LIN {X 0,Y 573.286,Z 217.077,A -85,B 0,C 180,E1 -2331.54,E2 -2331.54} C_VEL
LIN {X 0,Y 573.293,Z 217.075,A -85,B 0,C 180,E1 -2334.371,E2 -2334.371} C_VEL
LIN {X 0,Y 573.307,Z 217.075,A -85,B 0,C 180,E1 -2337.188,E2 -2337.188} C_VEL
LIN {X 0,Y 573.317,Z 217.072,A -85,B 0,C 180,E1 -2339.999,E2 -2339.999} C_VEL
LIN {X 0,Y 573.307,Z 217.074,A -85,B 0,C 180,E1 -2342.809,E2 -2342.809} C_VEL
LIN {X 0,Y 573.288,Z 217.076,A -85,B 0,C 180,E1 -2345.627,E2 -2345.627} C_VEL
LIN {X 0,Y 573.302,Z 217.075,A -85,B 0,C 180,E1 -2348.458,E2 -2348.458} C_VEL
LIN {X 0,Y 573.292,Z 217.075,A -85,B 0,C 180,E1 -2351.31,E2 -2351.31} C_VEL
LIN {X 0,Y 573.273,Z 217.08,A -85,B 0,C 180,E1 -2354.424,E2 -2354.424} C_VEL
LIN {X 0,Y 573.246,Z 217.081,A -85,B 0,C 180,E1 -2357.111,E2 -2357.111} C_VEL
LIN {X 0,Y 573.119,Z 217.099,A -85,B 0,C 180,E1 -2358.591,E2 -2358.591} C_VEL
LIN {X 0,Y 573.089,Z 220.567,A -85,B 0,C 180,E1 -2361.585,E2 -2361.585} C_VEL
LIN {X 0,Y 573.066,Z 223.811,A -85,B 0,C 180,E1 -2364.338,E2 -2364.338} C_VEL
LIN {X 0,Y 572.416,Z 224.562,A -85,B 0,C 180,E1 -2364.919,E2 -2364.919} C_VEL
LIN {X 0,Y 569.55,Z 225.938,A -85,B 0,C 180,E1 -2365.861,E2 -2365.861} C_VEL
LIN {X 0,Y 567.109,Z 227.058,A -85,B 0,C 180,E1 -2366.618,E2 -2366.618} C_VEL
LIN {X 0,Y 566.053,Z 227.855,A -85,B 0,C 180,E1 -2367.204,E2 -2367.204} C_VEL
LIN {X 0,Y 565.963,Z 228.105,A -85,B 0,C 180,E1 -2367.402,E2 -2367.402} C_VEL
LIN {X 0,Y 565.967,Z 230.788,A -85,B 0,C 180,E1 -2369.781,E2 -2369.781} C_VEL
LIN {X 0,Y 565.878,Z 233.608,A -85,B 0,C 180,E1 -2372.379,E2 -2372.379} C_VEL
LIN {X 0,Y 565.833,Z 236.534,A -85,B 0,C 180,E1 -2374.941,E2 -2374.941} C_VEL
LIN {X 0,Y 565.809,Z 239.829,A -85,B 0,C 180,E1 -2377.489,E2 -2377.489} C_VEL
LIN {X 0,Y 565.833,Z 243.678,A -85,B 0,C 180,E1 -2380.428,E2 -2380.428} C_VEL
LIN {X 0,Y 566.887,Z 251.297,A -85,B 0,C 180,E1 -2380.629,E2 -2380.629} C_VEL
LIN {X 0,Y 566.793,Z 264.173,A -85,B 0,C 180,E1 -2381.027,E2 -2381.027} C_VEL
LIN {X 0,Y 566.586,Z 276.718,A -85,B 0,C 180,E1 -2381.574,E2 -2381.574} C_VEL
LIN {X 0,Y 566.487,Z 287.395,A -85,B 0,C 180,E1 -2382.18,E2 -2382.18} C_VEL
LIN {X 0,Y 566.375,Z 298.091,A -85,B 0,C 180,E1 -2382.937,E2 -2382.937} C_VEL
LIN {X 0,Y 566.243,Z 307.919,A -85,B 0,C 180,E1 -2383.797,E2 -2383.797} C_VEL
LIN {X 0,Y 566.107,Z 317.442,A -85,B 0,C 180,E1 -2384.833,E2 -2384.833} C_VEL
LIN {X 0,Y 566.031,Z 325.716,A -85,B 0,C 180,E1 -2385.949,E2 -2385.949} C_VEL
LIN {X 0,Y 565.958,Z 332.481,A -85,B 0,C 180,E1 -2387.107,E2 -2387.107} C_VEL
LIN {X 0,Y 565.935,Z 337.377,A -85,B 0,C 180,E1 -2388.165,E2 -2388.165} C_VEL
LIN {X 0,Y 565.917,Z 341.246,A -85,B 0,C 180,E1 -2389.246,E2 -2389.246} C_VEL
LIN {X 0,Y 565.871,Z 344.136,A -85,B 0,C 180,E1 -2390.354,E2 -2390.354} C_VEL
LIN {X 0,Y 565.847,Z 346.173,A -85,B 0,C 180,E1 -2391.611,E2 -2391.611} C_VEL
LIN {X 0,Y 565.833,Z 346.918,A -85,B 0,C 180,E1 -2392.645,E2 -2392.645} C_VEL
LIN {X 0,Y 565.815,Z 346.733,A -85,B 0,C 180,E1 -2393.836,E2 -2393.836} C_VEL
LIN {X 0,Y 565.847,Z 345.233,A -85,B 0,C 180,E1 -2395.158,E2 -2395.158} C_VEL
LIN {X 0,Y 565.899,Z 342.77,A -85,B 0,C 180,E1 -2396.31,E2 -2396.31} C_VEL
LIN {X 0,Y 565.878,Z 338.598,A -85,B 0,C 180,E1 -2397.619,E2 -2397.619} C_VEL
LIN {X 0,Y 565.944,Z 334.577,A -85,B 0,C 180,E1 -2398.564,E2 -2398.564} C_VEL
LIN {X 0,Y 566.021,Z 329.055,A -85,B 0,C 180,E1 -2399.605,E2 -2399.605} C_VEL
LIN {X 0,Y 566.069,Z 322.304,A -85,B 0,C 180,E1 -2400.633,E2 -2400.633} C_VEL
LIN {X 0,Y 566.159,Z 313.851,A -85,B 0,C 180,E1 -2401.674,E2 -2401.674} C_VEL
LIN {X 0,Y 566.27,Z 303.926,A -85,B 0,C 180,E1 -2402.665,E2 -2402.665} C_VEL
LIN {X 0,Y 566.435,Z 293.893,A -85,B 0,C 180,E1 -2403.471,E2 -2403.471} C_VEL
LIN {X 0,Y 566.508,Z 283.157,A -85,B 0,C 180,E1 -2404.168,E2 -2404.168} C_VEL
LIN {X 0,Y 566.677,Z 271.149,A -85,B 0,C 180,E1 -2404.779,E2 -2404.779} C_VEL
LIN {X 0,Y 566.823,Z 259.841,A -85,B 0,C 180,E1 -2405.214,E2 -2405.214} C_VEL
LIN {X 0,Y 566.718,Z 248.791,A -85,B 0,C 180,E1 -2405.527,E2 -2405.527} C_VEL
LIN {X 0,Y 565.875,Z 243.68,A -85,B 0,C 180,E1 -2405.659,E2 -2405.659} C_VEL
LIN {X 0,Y 565.885,Z 239.45,A -85,B 0,C 180,E1 -2408.89,E2 -2408.89} C_VEL
LIN {X 0,Y 565.873,Z 236.517,A -85,B 0,C 180,E1 -2411.162,E2 -2411.162} C_VEL
LIN {X 0,Y 565.896,Z 233.864,A -85,B 0,C 180,E1 -2413.404,E2 -2413.404} C_VEL
LIN {X 0,Y 565.962,Z 230.528,A -85,B 0,C 180,E1 -2416.354,E2 -2416.354} C_VEL
LIN {X 0,Y 565.958,Z 227.036,A -85,B 0,C 180,E1 -2419.266,E2 -2419.266} C_VEL
LIN {X 0,Y 566.008,Z 223.617,A -85,B 0,C 180,E1 -2422.15,E2 -2422.15} C_VEL
LIN {X 0,Y 566.06,Z 220.337,A -85,B 0,C 180,E1 -2425.015,E2 -2425.015} C_VEL
LIN {X 0,Y 566.002,Z 217.986,A -85,B 0,C 180,E1 -2427.154,E2 -2427.154} C_VEL
LIN {X 0,Y 566.299,Z 217.947,A -85,B 0,C 180,E1 -2429.29,E2 -2429.29} C_VEL
LIN {X 0,Y 566.27,Z 217.949,A -85,B 0,C 180,E1 -2432.135,E2 -2432.135} C_VEL
LIN {X 0,Y 566.251,Z 217.952,A -85,B 0,C 180,E1 -2435.699,E2 -2435.699} C_VEL
LIN {X 0,Y 566.238,Z 217.955,A -85,B 0,C 180,E1 -2438.566,E2 -2438.566} C_VEL
LIN {X 0,Y 566.238,Z 217.953,A -85,B 0,C 180,E1 -2441.455,E2 -2441.455} C_VEL
LIN {X 0,Y 566.221,Z 217.957,A -85,B 0,C 180,E1 -2444.508,E2 -2444.508} C_VEL
LIN {X 0,Y 566.193,Z 217.959,A -85,B 0,C 180,E1 -2447.333,E2 -2447.333} C_VEL
LIN {X 0,Y 566.21,Z 217.958,A -85,B 0,C 180,E1 -2450.338,E2 -2450.338} C_VEL
LIN {X 0,Y 566.219,Z 217.958,A -85,B 0,C 180,E1 -2453.403,E2 -2453.403} C_VEL
LIN {X 0,Y 566.217,Z 217.958,A -85,B 0,C 180,E1 -2455.75,E2 -2455.75} C_VEL
LIN {X 0,Y 566.199,Z 217.96,A -85,B 0,C 180,E1 -2458.205,E2 -2458.205} C_VEL
LIN {X 0,Y 566.19,Z 217.96,A -85,B 0,C 180,E1 -2461.08,E2 -2461.08} C_VEL
LIN {X 0,Y 566.221,Z 217.958,A -85,B 0,C 180,E1 -2463.739,E2 -2463.739} C_VEL
LIN {X 0,Y 566.209,Z 217.957,A -85,B 0,C 180,E1 -2466.57,E2 -2466.57} C_VEL
LIN {X 0,Y 566.207,Z 217.959,A -85,B 0,C 180,E1 -2469.687,E2 -2469.687} C_VEL
LIN {X 0,Y 566.211,Z 217.958,A -85,B 0,C 180,E1 -2472.088,E2 -2472.088} C_VEL
LIN {X 0,Y 566.167,Z 217.964,A -85,B 0,C 180,E1 -2475.037,E2 -2475.037} C_VEL
LIN {X 0,Y 566.213,Z 217.956,A -85,B 0,C 180,E1 -2478.137,E2 -2478.137} C_VEL
LIN {X 0,Y 566.22,Z 217.957,A -85,B 0,C 180,E1 -2480.729,E2 -2480.729} C_VEL
LIN {X 0,Y 566.212,Z 217.956,A -85,B 0,C 180,E1 -2483.785,E2 -2483.785} C_VEL
LIN {X 0,Y 566.227,Z 217.955,A -85,B 0,C 180,E1 -2486.9,E2 -2486.9} C_VEL
LIN {X 0,Y 566.18,Z 217.96,A -85,B 0,C 180,E1 -2489.409,E2 -2489.409} C_VEL
LIN {X 0,Y 566.211,Z 217.957,A -85,B 0,C 180,E1 -2491.859,E2 -2491.859} C_VEL
LIN {X 0,Y 566.215,Z 217.956,A -85,B 0,C 180,E1 -2494.253,E2 -2494.253} C_VEL
LIN {X 0,Y 566.17,Z 217.963,A -85,B 0,C 180,E1 -2496.721,E2 -2496.721} C_VEL
LIN {X 0,Y 566.217,Z 217.956,A -85,B 0,C 180,E1 -2499.664,E2 -2499.664} C_VEL
LIN {X 0,Y 566.202,Z 217.96,A -85,B 0,C 180,E1 -2502.67,E2 -2502.67} C_VEL
LIN {X 0,Y 566.238,Z 217.953,A -85,B 0,C 180,E1 -2505.628,E2 -2505.628} C_VEL
LIN {X 0,Y 566.239,Z 217.953,A -85,B 0,C 180,E1 -2508.677,E2 -2508.677} C_VEL
LIN {X 0,Y 566.211,Z 217.957,A -85,B 0,C 180,E1 -2511.435,E2 -2511.435} C_VEL
LIN {X 0,Y 566.216,Z 217.956,A -85,B 0,C 180,E1 -2513.587,E2 -2513.587} C_VEL
LIN {X 0,Y 566.187,Z 217.96,A -85,B 0,C 180,E1 -2515.73,E2 -2515.73} C_VEL
LIN {X 0,Y 566.276,Z 217.949,A -85,B 0,C 180,E1 -2517.867,E2 -2517.867} C_VEL
LIN {X 0,Y 566.302,Z 217.946,A -85,B 0,C 180,E1 -2520.712,E2 -2520.712} C_VEL
LIN {X 0,Y 566.271,Z 217.948,A -85,B 0,C 180,E1 -2522.847,E2 -2522.847} C_VEL
LIN {X 0,Y 566.258,Z 217.953,A -85,B 0,C 180,E1 -2525.699,E2 -2525.699} C_VEL
LIN {X 0,Y 566.212,Z 217.956,A -85,B 0,C 180,E1 -2528.567,E2 -2528.567} C_VEL
LIN {X 0,Y 566.25,Z 217.954,A -85,B 0,C 180,E1 -2531.455,E2 -2531.455} C_VEL
LIN {X 0,Y 566.227,Z 217.955,A -85,B 0,C 180,E1 -2534.501,E2 -2534.501} C_VEL
LIN {X 0,Y 566.198,Z 217.959,A -85,B 0,C 180,E1 -2537.333,E2 -2537.333} C_VEL
LIN {X 0,Y 566.216,Z 217.958,A -85,B 0,C 180,E1 -2540.338,E2 -2540.338} C_VEL
LIN {X 0,Y 566.175,Z 217.961,A -85,B 0,C 180,E1 -2543.281,E2 -2543.281} C_VEL
LIN {X 0,Y 566.211,Z 217.957,A -85,B 0,C 180,E1 -2545.75,E2 -2545.75} C_VEL
LIN {X 0,Y 566.212,Z 217.957,A -85,B 0,C 180,E1 -2548.202,E2 -2548.202} C_VEL
LIN {X 0,Y 566.194,Z 217.96,A -85,B 0,C 180,E1 -2551.076,E2 -2551.076} C_VEL
LIN {X 0,Y 566.205,Z 217.957,A -85,B 0,C 180,E1 -2553.732,E2 -2553.732} C_VEL
LIN {X 0,Y 566.208,Z 217.96,A -85,B 0,C 180,E1 -2556.57,E2 -2556.57} C_VEL
LIN {X 0,Y 566.221,Z 217.957,A -85,B 0,C 180,E1 -2559.686,E2 -2559.686} C_VEL
LIN {X 0,Y 566.21,Z 217.957,A -85,B 0,C 180,E1 -2562.917,E2 -2562.917} C_VEL
LIN {X 0,Y 566.202,Z 217.957,A -85,B 0,C 180,E1 -2566.049,E2 -2566.049} C_VEL
LIN {X 0,Y 566.212,Z 217.958,A -85,B 0,C 180,E1 -2569.214,E2 -2569.214} C_VEL
LIN {X 0,Y 566.189,Z 217.962,A -85,B 0,C 180,E1 -2571.636,E2 -2571.636} C_VEL
LIN {X 0,Y 566.229,Z 218.104,A -85,B 0,C 180,E1 -2573.043,E2 -2573.043} C_VEL
LIN {X 0,Y 566.784,Z 221.774,A -85,B 0,C 180,E1 -2574.352,E2 -2574.352} C_VEL
LIN {X 0,Y 566.714,Z 229.498,A -85,B 0,C 180,E1 -2576.93,E2 -2576.93} C_VEL
LIN {X 0,Y 566.515,Z 237.229,A -85,B 0,C 180,E1 -2579.426,E2 -2579.426} C_VEL
LIN {X 0,Y 566.446,Z 245.3,A -85,B 0,C 180,E1 -2581.869,E2 -2581.869} C_VEL
LIN {X 0,Y 566.345,Z 255.739,A -85,B 0,C 180,E1 -2584.944,E2 -2584.944} C_VEL
LIN {X 0,Y 566.292,Z 265.468,A -85,B 0,C 180,E1 -2587.757,E2 -2587.757} C_VEL
LIN {X 0,Y 566.209,Z 275.582,A -85,B 0,C 180,E1 -2590.622,E2 -2590.622} C_VEL
LIN {X 0,Y 566.129,Z 285.461,A -85,B 0,C 180,E1 -2593.409,E2 -2593.409} C_VEL
LIN {X 0,Y 566.046,Z 296.052,A -85,B 0,C 180,E1 -2596.354,E2 -2596.354} C_VEL
LIN {X 0,Y 566.015,Z 299.528,A -85,B 0,C 180,E1 -2597.313,E2 -2597.313} C_VEL
LIN {X 0,Y 566.935,Z 306.333,A -85,B 0,C 180,E1 -2597.47,E2 -2597.47} C_VEL
LIN {X 0,Y 566.844,Z 318.476,A -85,B 0,C 180,E1 -2597.786,E2 -2597.786} C_VEL
LIN {X 0,Y 566.689,Z 330.299,A -85,B 0,C 180,E1 -2598.228,E2 -2598.228} C_VEL
LIN {X 0,Y 566.534,Z 342.971,A -85,B 0,C 180,E1 -2598.867,E2 -2598.867} C_VEL
LIN {X 0,Y 566.439,Z 354.736,A -85,B 0,C 180,E1 -2599.635,E2 -2599.635} C_VEL
LIN {X 0,Y 566.302,Z 363.639,A -85,B 0,C 180,E1 -2600.355,E2 -2600.355} C_VEL
LIN {X 0,Y 566.162,Z 372.78,A -85,B 0,C 180,E1 -2601.253,E2 -2601.253} C_VEL
LIN {X 0,Y 566.082,Z 381.684,A -85,B 0,C 180,E1 -2602.33,E2 -2602.33} C_VEL
LIN {X 0,Y 565.969,Z 388.952,A -85,B 0,C 180,E1 -2603.422,E2 -2603.422} C_VEL
LIN {X 0,Y 566.004,Z 393.676,A -85,B 0,C 180,E1 -2604.298,E2 -2604.298} C_VEL
LIN {X 0,Y 565.933,Z 398.369,A -85,B 0,C 180,E1 -2605.369,E2 -2605.369} C_VEL
LIN {X 0,Y 565.927,Z 401.956,A -85,B 0,C 180,E1 -2606.439,E2 -2606.439} C_VEL
LIN {X 0,Y 565.878,Z 403.806,A -85,B 0,C 180,E1 -2607.152,E2 -2607.152} C_VEL
LIN {X 0,Y 565.846,Z 406.184,A -85,B 0,C 180,E1 -2608.576,E2 -2608.576} C_VEL
LIN {X 0,Y 565.839,Z 407,A -85,B 0,C 180,E1 -2609.999,E2 -2609.999} C_VEL
LIN {X 0,Y 565.846,Z 406.187,A -85,B 0,C 180,E1 -2611.423,E2 -2611.423} C_VEL
LIN {X 0,Y 565.878,Z 403.812,A -85,B 0,C 180,E1 -2612.847,E2 -2612.847} C_VEL
LIN {X 0,Y 565.926,Z 400.898,A -85,B 0,C 180,E1 -2613.916,E2 -2613.916} C_VEL
LIN {X 0,Y 565.878,Z 396.952,A -85,B 0,C 180,E1 -2614.987,E2 -2614.987} C_VEL
LIN {X 0,Y 566.002,Z 391.871,A -85,B 0,C 180,E1 -2616.058,E2 -2616.058} C_VEL
LIN {X 0,Y 566.04,Z 385.473,A -85,B 0,C 180,E1 -2617.132,E2 -2617.132} C_VEL
LIN {X 0,Y 566.133,Z 377.484,A -85,B 0,C 180,E1 -2618.207,E2 -2618.207} C_VEL
LIN {X 0,Y 566.229,Z 369.342,A -85,B 0,C 180,E1 -2619.105,E2 -2619.105} C_VEL
LIN {X 0,Y 566.348,Z 359.409,A -85,B 0,C 180,E1 -2620.004,E2 -2620.004} C_VEL
LIN {X 0,Y 566.502,Z 348.334,A -85,B 0,C 180,E1 -2620.805,E2 -2620.805} C_VEL
LIN {X 0,Y 566.608,Z 335.96,A -85,B 0,C 180,E1 -2621.509,E2 -2621.509} C_VEL
LIN {X 0,Y 566.749,Z 323.789,A -85,B 0,C 180,E1 -2622.033,E2 -2622.033} C_VEL
LIN {X 0,Y 566.928,Z 310.377,A -85,B 0,C 180,E1 -2622.438,E2 -2622.438} C_VEL
LIN {X 0,Y 566.641,Z 303.554,A -85,B 0,C 180,E1 -2622.592,E2 -2622.592} C_VEL
LIN {X 0,Y 566.014,Z 299.533,A -85,B 0,C 180,E1 -2622.686,E2 -2622.686} C_VEL
LIN {X 0,Y 566.089,Z 289.438,A -85,B 0,C 180,E1 -2625.48,E2 -2625.48} C_VEL
LIN {X 0,Y 566.175,Z 278.847,A -85,B 0,C 180,E1 -2628.453,E2 -2628.453} C_VEL
LIN {X 0,Y 566.237,Z 269.442,A -85,B 0,C 180,E1 -2631.096,E2 -2631.096} C_VEL
LIN {X 0,Y 566.278,Z 259.722,A -85,B 0,C 180,E1 -2633.787,E2 -2633.787} C_VEL
LIN {X 0,Y 566.331,Z 250.15,A -85,B 0,C 180,E1 -2636.534,E2 -2636.534} C_VEL
LIN {X 0,Y 566.468,Z 241.095,A -85,B 0,C 180,E1 -2639.33,E2 -2639.33} C_VEL
LIN {X 0,Y 566.63,Z 231.929,A -85,B 0,C 180,E1 -2642.23,E2 -2642.23} C_VEL
LIN {X 0,Y 566.775,Z 224.253,A -85,B 0,C 180,E1 -2644.777,E2 -2644.777} C_VEL
LIN {X 0,Y 566.551,Z 220.044,A -85,B 0,C 180,E1 -2646.261,E2 -2646.261} C_VEL
LIN {X 0,Y 566.205,Z 217.959,A -85,B 0,C 180,E1 -2647.109,E2 -2647.109} C_VEL
LIN {X 0,Y 566.212,Z 217.959,A -85,B 0,C 180,E1 -2649.685,E2 -2649.685} C_VEL
LIN {X 0,Y 566.214,Z 217.959,A -85,B 0,C 180,E1 -2652.086,E2 -2652.086} C_VEL
LIN {X 0,Y 566.167,Z 217.963,A -85,B 0,C 180,E1 -2655.035,E2 -2655.035} C_VEL
LIN {X 0,Y 566.218,Z 217.956,A -85,B 0,C 180,E1 -2658.135,E2 -2658.135} C_VEL
LIN {X 0,Y 566.215,Z 217.957,A -85,B 0,C 180,E1 -2660.726,E2 -2660.726} C_VEL
LIN {X 0,Y 566.202,Z 217.958,A -85,B 0,C 180,E1 -2663.784,E2 -2663.784} C_VEL
LIN {X 0,Y 566.211,Z 217.957,A -85,B 0,C 180,E1 -2666.265,E2 -2666.265} C_VEL
LIN {X 0,Y 566.187,Z 217.962,A -85,B 0,C 180,E1 -2668.923,E2 -2668.923} C_VEL
LIN {X 0,Y 566.226,Z 217.955,A -85,B 0,C 180,E1 -2671.857,E2 -2671.857} C_VEL
LIN {X 0,Y 566.212,Z 217.957,A -85,B 0,C 180,E1 -2674.25,E2 -2674.25} C_VEL
LIN {X 0,Y 566.166,Z 217.963,A -85,B 0,C 180,E1 -2676.718,E2 -2676.718} C_VEL
LIN {X 0,Y 566.211,Z 217.957,A -85,B 0,C 180,E1 -2679.662,E2 -2679.662} C_VEL
LIN {X 0,Y 566.197,Z 217.961,A -85,B 0,C 180,E1 -2682.667,E2 -2682.667} C_VEL
LIN {X 0,Y 566.231,Z 217.954,A -85,B 0,C 180,E1 -2685.626,E2 -2685.626} C_VEL
LIN {X 0,Y 566.23,Z 217.954,A -85,B 0,C 180,E1 -2688.674,E2 -2688.674} C_VEL
LIN {X 0,Y 566.229,Z 217.955,A -85,B 0,C 180,E1 -2691.433,E2 -2691.433} C_VEL
LIN {X 0,Y 566.26,Z 217.951,A -85,B 0,C 180,E1 -2694.301,E2 -2694.301} C_VEL
LIN {X 0,Y 566.271,Z 217.949,A -85,B 0,C 180,E1 -2697.865,E2 -2697.865} C_VEL
LIN {X 0,Y 566.304,Z 217.948,A -85,B 0,C 180,E1 -2700.71,E2 -2700.71} C_VEL
LIN {X 0,Y 566.272,Z 217.951,A -85,B 0,C 180,E1 -2702.844,E2 -2702.844} C_VEL
LIN {X 0,Y 566.256,Z 217.951,A -85,B 0,C 180,E1 -2705.697,E2 -2705.697} C_VEL
LIN {X 0,Y 566.243,Z 217.955,A -85,B 0,C 180,E1 -2708.564,E2 -2708.564} C_VEL
LIN {X 0,Y 566.244,Z 217.953,A -85,B 0,C 180,E1 -2711.453,E2 -2711.453} C_VEL
LIN {X 0,Y 566.226,Z 217.957,A -85,B 0,C 180,E1 -2714.506,E2 -2714.506} C_VEL
LIN {X 0,Y 566.178,Z 217.962,A -85,B 0,C 180,E1 -2717.331,E2 -2717.331} C_VEL
LIN {X 0,Y 566.055,Z 218.047,A -85,B 0,C 180,E1 -2718.831,E2 -2718.831} C_VEL
LIN {X 0,Y 566.049,Z 220.993,A -85,B 0,C 180,E1 -2721.381,E2 -2721.381} C_VEL
LIN {X 0,Y 565.99,Z 224.427,A -85,B 0,C 180,E1 -2724.331,E2 -2724.331} C_VEL
LIN {X 0,Y 565.985,Z 227.149,A -85,B 0,C 180,E1 -2726.616,E2 -2726.616} C_VEL
LIN {X 0,Y 565.963,Z 228.105,A -85,B 0,C 180,E1 -2727.402,E2 -2727.402} C_VEL
LIN {X 0,Y 565.283,Z 228.882,A -85,B 0,C 180,E1 -2727.991,E2 -2727.991} C_VEL
LIN {X 0,Y 562.408,Z 230.258,A -85,B 0,C 180,E1 -2728.946,E2 -2728.946} C_VEL
LIN {X 0,Y 559.98,Z 231.306,A -85,B 0,C 180,E1 -2729.715,E2 -2729.715} C_VEL
LIN {X 0,Y 558.934,Z 232.024,A -85,B 0,C 180,E1 -2730.31,E2 -2730.31} C_VEL
LIN {X 0,Y 558.847,Z 232.245,A -85,B 0,C 180,E1 -2730.511,E2 -2730.511} C_VEL
LIN {X 0,Y 558.809,Z 235.592,A -85,B 0,C 180,E1 -2733.597,E2 -2733.597} C_VEL
LIN {X 0,Y 558.731,Z 238.749,A -85,B 0,C 180,E1 -2736.389,E2 -2736.389} C_VEL
LIN {X 0,Y 558.713,Z 241.999,A -85,B 0,C 180,E1 -2738.97,E2 -2738.97} C_VEL
LIN {X 0,Y 558.751,Z 243.681,A -85,B 0,C 180,E1 -2740.268,E2 -2740.268} C_VEL
LIN {X 0,Y 559.962,Z 252.449,A -85,B 0,C 180,E1 -2740.502,E2 -2740.502} C_VEL
LIN {X 0,Y 559.843,Z 264.145,A -85,B 0,C 180,E1 -2740.874,E2 -2740.874} C_VEL
LIN {X 0,Y 559.631,Z 276.024,A -85,B 0,C 180,E1 -2741.394,E2 -2741.394} C_VEL
LIN {X 0,Y 559.492,Z 288.404,A -85,B 0,C 180,E1 -2742.107,E2 -2742.107} C_VEL
LIN {X 0,Y 559.361,Z 298.544,A -85,B 0,C 180,E1 -2742.845,E2 -2742.845} C_VEL
LIN {X 0,Y 559.202,Z 308.372,A -85,B 0,C 180,E1 -2743.726,E2 -2743.726} C_VEL
LIN {X 0,Y 559.064,Z 317.573,A -85,B 0,C 180,E1 -2744.745,E2 -2744.745} C_VEL
LIN {X 0,Y 558.978,Z 325.16,A -85,B 0,C 180,E1 -2745.777,E2 -2745.777} C_VEL
LIN {X 0,Y 558.88,Z 332.471,A -85,B 0,C 180,E1 -2747.029,E2 -2747.029} C_VEL
LIN {X 0,Y 558.838,Z 337.762,A -85,B 0,C 180,E1 -2748.201,E2 -2748.201} C_VEL
LIN {X 0,Y 558.825,Z 341.134,A -85,B 0,C 180,E1 -2749.159,E2 -2749.159} C_VEL
LIN {X 0,Y 558.785,Z 343.669,A -85,B 0,C 180,E1 -2750.102,E2 -2750.102} C_VEL
LIN {X 0,Y 558.741,Z 345.757,A -85,B 0,C 180,E1 -2751.244,E2 -2751.244} C_VEL
LIN {X 0,Y 558.74,Z 346.842,A -85,B 0,C 180,E1 -2752.411,E2 -2752.411} C_VEL
LIN {X 0,Y 558.719,Z 346.79,A -85,B 0,C 180,E1 -2753.759,E2 -2753.759} C_VEL
LIN {X 0,Y 558.746,Z 345.764,A -85,B 0,C 180,E1 -2754.84,E2 -2754.84} C_VEL
LIN {X 0,Y 558.793,Z 343.38,A -85,B 0,C 180,E1 -2756.105,E2 -2756.105} C_VEL
LIN {X 0,Y 558.788,Z 339.514,A -85,B 0,C 180,E1 -2757.42,E2 -2757.42} C_VEL
LIN {X 0,Y 558.848,Z 335.296,A -85,B 0,C 180,E1 -2758.473,E2 -2758.473} C_VEL
LIN {X 0,Y 558.935,Z 329.569,A -85,B 0,C 180,E1 -2759.597,E2 -2759.597} C_VEL
LIN {X 0,Y 558.988,Z 322.953,A -85,B 0,C 180,E1 -2760.638,E2 -2760.638} C_VEL
LIN {X 0,Y 559.093,Z 314.66,A -85,B 0,C 180,E1 -2761.693,E2 -2761.693} C_VEL
LIN {X 0,Y 559.238,Z 304.878,A -85,B 0,C 180,E1 -2762.698,E2 -2762.698} C_VEL
LIN {X 0,Y 559.425,Z 295.081,A -85,B 0,C 180,E1 -2763.515,E2 -2763.515} C_VEL
LIN {X 0,Y 559.522,Z 284.646,A -85,B 0,C 180,E1 -2764.221,E2 -2764.221} C_VEL
LIN {X 0,Y 559.711,Z 272.626,A -85,B 0,C 180,E1 -2764.858,E2 -2764.858} C_VEL
LIN {X 0,Y 559.877,Z 260.858,A -85,B 0,C 180,E1 -2765.332,E2 -2765.332} C_VEL
LIN {X 0,Y 559.73,Z 249.375,A -85,B 0,C 180,E1 -2765.671,E2 -2765.671} C_VEL
LIN {X 0,Y 558.776,Z 243.677,A -85,B 0,C 180,E1 -2765.824,E2 -2765.824} C_VEL
LIN {X 0,Y 558.764,Z 240.078,A -85,B 0,C 180,E1 -2768.608,E2 -2768.608} C_VEL
LIN {X 0,Y 558.805,Z 237.294,A -85,B 0,C 180,E1 -2770.914,E2 -2770.914} C_VEL
LIN {X 0,Y 558.831,Z 234.671,A -85,B 0,C 180,E1 -2773.188,E2 -2773.188} C_VEL
LIN {X 0,Y 558.891,Z 231.28,A -85,B 0,C 180,E1 -2776.178,E2 -2776.178} C_VEL
LIN {X 0,Y 558.904,Z 227.787,A -85,B 0,C 180,E1 -2779.129,E2 -2779.129} C_VEL
LIN {X 0,Y 558.936,Z 224.358,A -85,B 0,C 180,E1 -2782.051,E2 -2782.051} C_VEL
LIN {X 0,Y 559.004,Z 221.058,A -85,B 0,C 180,E1 -2784.952,E2 -2784.952} C_VEL
LIN {X 0,Y 558.933,Z 219.387,A -85,B 0,C 180,E1 -2786.396,E2 -2786.396} C_VEL
LIN {X 0,Y 558.949,Z 218.865,A -85,B 0,C 180,E1 -2787.118,E2 -2787.118} C_VEL
LIN {X 0,Y 559.158,Z 218.836,A -85,B 0,C 180,E1 -2788.56,E2 -2788.56} C_VEL
LIN {X 0,Y 559.268,Z 218.824,A -85,B 0,C 180,E1 -2790.721,E2 -2790.721} C_VEL
LIN {X 0,Y 559.229,Z 218.829,A -85,B 0,C 180,E1 -2792.882,E2 -2792.882} C_VEL
LIN {X 0,Y 559.22,Z 218.827,A -85,B 0,C 180,E1 -2795.771,E2 -2795.771} C_VEL
LIN {X 0,Y 559.193,Z 218.834,A -85,B 0,C 180,E1 -2798.675,E2 -2798.675} C_VEL
LIN {X 0,Y 559.196,Z 218.831,A -85,B 0,C 180,E1 -2801.601,E2 -2801.601} C_VEL
LIN {X 0,Y 559.186,Z 218.833,A -85,B 0,C 180,E1 -2804.597,E2 -2804.597} C_VEL
LIN {X 0,Y 559.152,Z 218.837,A -85,B 0,C 180,E1 -2807.558,E2 -2807.558} C_VEL
LIN {X 0,Y 559.164,Z 218.836,A -85,B 0,C 180,E1 -2809.838,E2 -2809.838} C_VEL
LIN {X 0,Y 559.145,Z 218.838,A -85,B 0,C 180,E1 -2812.153,E2 -2812.153} C_VEL
LIN {X 0,Y 559.149,Z 218.838,A -85,B 0,C 180,E1 -2814.506,E2 -2814.506} C_VEL
LIN {X 0,Y 559.171,Z 218.837,A -85,B 0,C 180,E1 -2816.903,E2 -2816.903} C_VEL
LIN {X 0,Y 559.14,Z 218.837,A -85,B 0,C 180,E1 -2819.859,E2 -2819.859} C_VEL
LIN {X 0,Y 559.167,Z 218.837,A -85,B 0,C 180,E1 -2822.715,E2 -2822.715} C_VEL
LIN {X 0,Y 559.151,Z 218.836,A -85,B 0,C 180,E1 -2825.323,E2 -2825.323} C_VEL
LIN {X 0,Y 559.127,Z 218.839,A -85,B 0,C 180,E1 -2828.019,E2 -2828.019} C_VEL
LIN {X 0,Y 559.17,Z 218.835,A -85,B 0,C 180,E1 -2830.812,E2 -2830.812} C_VEL
LIN {X 0,Y 559.158,Z 218.835,A -85,B 0,C 180,E1 -2833.733,E2 -2833.733} C_VEL
LIN {X 0,Y 559.141,Z 218.838,A -85,B 0,C 180,E1 -2836.805,E2 -2836.805} C_VEL
LIN {X 0,Y 559.172,Z 218.833,A -85,B 0,C 180,E1 -2839.191,E2 -2839.191} C_VEL
LIN {X 0,Y 559.132,Z 218.84,A -85,B 0,C 180,E1 -2841.984,E2 -2841.984} C_VEL
LIN {X 0,Y 559.147,Z 218.837,A -85,B 0,C 180,E1 -2844.786,E2 -2844.786} C_VEL
LIN {X 0,Y 559.171,Z 218.833,A -85,B 0,C 180,E1 -2847.363,E2 -2847.363} C_VEL
LIN {X 0,Y 559.148,Z 218.839,A -85,B 0,C 180,E1 -2850.144,E2 -2850.144} C_VEL
LIN {X 0,Y 559.169,Z 218.833,A -85,B 0,C 180,E1 -2853.099,E2 -2853.099} C_VEL
LIN {X 0,Y 559.156,Z 218.835,A -85,B 0,C 180,E1 -2855.496,E2 -2855.496} C_VEL
LIN {X 0,Y 559.174,Z 218.833,A -85,B 0,C 180,E1 -2858.625,E2 -2858.625} C_VEL
LIN {X 0,Y 559.169,Z 218.833,A -85,B 0,C 180,E1 -2860.928,E2 -2860.928} C_VEL
LIN {X 0,Y 559.165,Z 218.837,A -85,B 0,C 180,E1 -2863.949,E2 -2863.949} C_VEL
LIN {X 0,Y 559.175,Z 218.836,A -85,B 0,C 180,E1 -2866.186,E2 -2866.186} C_VEL
LIN {X 0,Y 559.197,Z 218.83,A -85,B 0,C 180,E1 -2869.135,E2 -2869.135} C_VEL
LIN {X 0,Y 559.196,Z 218.832,A -85,B 0,C 180,E1 -2872.055,E2 -2872.055} C_VEL
LIN {X 0,Y 559.256,Z 218.823,A -85,B 0,C 180,E1 -2874.955,E2 -2874.955} C_VEL
LIN {X 0,Y 559.249,Z 218.825,A -85,B 0,C 180,E1 -2877.841,E2 -2877.841} C_VEL
LIN {X 0,Y 559.273,Z 218.821,A -85,B 0,C 180,E1 -2880.721,E2 -2880.721} C_VEL
LIN {X 0,Y 559.239,Z 218.824,A -85,B 0,C 180,E1 -2882.882,E2 -2882.882} C_VEL
LIN {X 0,Y 559.228,Z 218.828,A -85,B 0,C 180,E1 -2885.771,E2 -2885.771} C_VEL
LIN {X 0,Y 559.176,Z 218.833,A -85,B 0,C 180,E1 -2888.676,E2 -2888.676} C_VEL
LIN {X 0,Y 559.213,Z 218.829,A -85,B 0,C 180,E1 -2891.601,E2 -2891.601} C_VEL
LIN {X 0,Y 559.19,Z 218.833,A -85,B 0,C 180,E1 -2894.588,E2 -2894.588} C_VEL
LIN {X 0,Y 559.143,Z 218.837,A -85,B 0,C 180,E1 -2897.558,E2 -2897.558} C_VEL
LIN {X 0,Y 559.175,Z 218.833,A -85,B 0,C 180,E1 -2899.838,E2 -2899.838} C_VEL
LIN {X 0,Y 559.148,Z 218.836,A -85,B 0,C 180,E1 -2902.153,E2 -2902.153} C_VEL
LIN {X 0,Y 559.148,Z 218.838,A -85,B 0,C 180,E1 -2905.178,E2 -2905.178} C_VEL
LIN {X 0,Y 559.15,Z 218.836,A -85,B 0,C 180,E1 -2907.715,E2 -2907.715} C_VEL
LIN {X 0,Y 559.157,Z 218.834,A -85,B 0,C 180,E1 -2910.183,E2 -2910.183} C_VEL
LIN {X 0,Y 559.159,Z 218.835,A -85,B 0,C 180,E1 -2912.716,E2 -2912.716} C_VEL
LIN {X 0,Y 559.136,Z 218.841,A -85,B 0,C 180,E1 -2915.324,E2 -2915.324} C_VEL
LIN {X 0,Y 559.138,Z 218.837,A -85,B 0,C 180,E1 -2918.018,E2 -2918.018} C_VEL
LIN {X 0,Y 559.164,Z 218.835,A -85,B 0,C 180,E1 -2920.813,E2 -2920.813} C_VEL
LIN {X 0,Y 559.146,Z 218.837,A -85,B 0,C 180,E1 -2923.734,E2 -2923.734} C_VEL
LIN {X 0,Y 559.153,Z 218.838,A -85,B 0,C 180,E1 -2926.804,E2 -2926.804} C_VEL
LIN {X 0,Y 559.164,Z 218.836,A -85,B 0,C 180,E1 -2929.187,E2 -2929.187} C_VEL
LIN {X 0,Y 559.137,Z 218.839,A -85,B 0,C 180,E1 -2931.982,E2 -2931.982} C_VEL
LIN {X 0,Y 559.162,Z 218.929,A -85,B 0,C 180,E1 -2932.795,E2 -2932.795} C_VEL
LIN {X 0,Y 559.821,Z 223.042,A -85,B 0,C 180,E1 -2934.284,E2 -2934.284} C_VEL
LIN {X 0,Y 559.741,Z 230.761,A -85,B 0,C 180,E1 -2936.894,E2 -2936.894} C_VEL
LIN {X 0,Y 559.537,Z 238.487,A -85,B 0,C 180,E1 -2939.422,E2 -2939.422} C_VEL
LIN {X 0,Y 559.43,Z 246.661,A -85,B 0,C 180,E1 -2941.933,E2 -2941.933} C_VEL
LIN {X 0,Y 559.345,Z 256.197,A -85,B 0,C 180,E1 -2944.778,E2 -2944.778} C_VEL
LIN {X 0,Y 559.217,Z 265.249,A -85,B 0,C 180,E1 -2947.46,E2 -2947.46} C_VEL
LIN {X 0,Y 559.147,Z 274.67,A -85,B 0,C 180,E1 -2950.161,E2 -2950.161} C_VEL
LIN {X 0,Y 559.083,Z 284.139,A -85,B 0,C 180,E1 -2952.818,E2 -2952.818} C_VEL
LIN {X 0,Y 558.986,Z 293.602,A -85,B 0,C 180,E1 -2955.491,E2 -2955.491} C_VEL
LIN {X 0,Y 558.94,Z 299.528,A -85,B 0,C 180,E1 -2957.149,E2 -2957.149} C_VEL
LIN {X 0,Y 560.017,Z 307.473,A -85,B 0,C 180,E1 -2957.336,E2 -2957.336} C_VEL
LIN {X 0,Y 559.878,Z 319.854,A -85,B 0,C 180,E1 -2957.678,E2 -2957.678} C_VEL
LIN {X 0,Y 559.725,Z 332.265,A -85,B 0,C 180,E1 -2958.17,E2 -2958.17} C_VEL
LIN {X 0,Y 559.558,Z 343.762,A -85,B 0,C 180,E1 -2958.773,E2 -2958.773} C_VEL
LIN {X 0,Y 559.428,Z 354.735,A -85,B 0,C 180,E1 -2959.504,E2 -2959.504} C_VEL
LIN {X 0,Y 559.245,Z 365.592,A -85,B 0,C 180,E1 -2960.414,E2 -2960.414} C_VEL
LIN {X 0,Y 559.123,Z 374.406,A -85,B 0,C 180,E1 -2961.324,E2 -2961.324} C_VEL
LIN {X 0,Y 558.998,Z 382.997,A -85,B 0,C 180,E1 -2962.413,E2 -2962.413} C_VEL
LIN {X 0,Y 558.886,Z 390.686,A -85,B 0,C 180,E1 -2963.649,E2 -2963.649} C_VEL
LIN {X 0,Y 558.869,Z 395.363,A -85,B 0,C 180,E1 -2964.587,E2 -2964.587} C_VEL
LIN {X 0,Y 558.869,Z 399.675,A -85,B 0,C 180,E1 -2965.672,E2 -2965.672} C_VEL
LIN {X 0,Y 558.837,Z 401.956,A -85,B 0,C 180,E1 -2966.394,E2 -2966.394} C_VEL
LIN {X 0,Y 558.8,Z 403.806,A -85,B 0,C 180,E1 -2967.116,E2 -2967.116} C_VEL
LIN {X 0,Y 558.745,Z 406.183,A -85,B 0,C 180,E1 -2968.558,E2 -2968.558} C_VEL
LIN {X 0,Y 558.74,Z 407,A -85,B 0,C 180,E1 -2969.999,E2 -2969.999} C_VEL
LIN {X 0,Y 558.745,Z 406.186,A -85,B 0,C 180,E1 -2971.441,E2 -2971.441} C_VEL
LIN {X 0,Y 558.799,Z 403.812,A -85,B 0,C 180,E1 -2972.883,E2 -2972.883} C_VEL
LIN {X 0,Y 558.844,Z 400.898,A -85,B 0,C 180,E1 -2973.965,E2 -2973.965} C_VEL
LIN {X 0,Y 558.798,Z 396.951,A -85,B 0,C 180,E1 -2975.05,E2 -2975.05} C_VEL
LIN {X 0,Y 558.918,Z 391.871,A -85,B 0,C 180,E1 -2976.135,E2 -2976.135} C_VEL
LIN {X 0,Y 558.977,Z 385.473,A -85,B 0,C 180,E1 -2977.222,E2 -2977.222} C_VEL
LIN {X 0,Y 559.099,Z 377.484,A -85,B 0,C 180,E1 -2978.311,E2 -2978.311} C_VEL
LIN {X 0,Y 559.195,Z 369.342,A -85,B 0,C 180,E1 -2979.22,E2 -2979.22} C_VEL
LIN {X 0,Y 559.362,Z 359.408,A -85,B 0,C 180,E1 -2980.13,E2 -2980.13} C_VEL
LIN {X 0,Y 559.506,Z 348.44,A -85,B 0,C 180,E1 -2980.935,E2 -2980.935} C_VEL
LIN {X 0,Y 559.636,Z 336.832,A -85,B 0,C 180,E1 -2981.609,E2 -2981.609} C_VEL
LIN {X 0,Y 559.791,Z 324.999,A -85,B 0,C 180,E1 -2982.138,E2 -2982.138} C_VEL
LIN {X 0,Y 559.991,Z 312.205,A -85,B 0,C 180,E1 -2982.548,E2 -2982.548} C_VEL
LIN {X 0,Y 559.816,Z 304.977,A -85,B 0,C 180,E1 -2982.719,E2 -2982.719} C_VEL
LIN {X 0,Y 558.938,Z 299.533,A -85,B 0,C 180,E1 -2982.849,E2 -2982.849} C_VEL
LIN {X 0,Y 559.054,Z 289.438,A -85,B 0,C 180,E1 -2985.68,E2 -2985.68} C_VEL
LIN {X 0,Y 559.141,Z 278.77,A -85,B 0,C 180,E1 -2988.693,E2 -2988.693} C_VEL
LIN {X 0,Y 559.173,Z 268.467,A -85,B 0,C 180,E1 -2991.553,E2 -2991.553} C_VEL
LIN {X 0,Y 559.225,Z 257.981,A -85,B 0,C 180,E1 -2994.501,E2 -2994.501} C_VEL
LIN {X 0,Y 559.328,Z 248.774,A -85,B 0,C 180,E1 -2997.298,E2 -2997.298} C_VEL
LIN {X 0,Y 559.504,Z 239.612,A -85,B 0,C 180,E1 -3000.161,E2 -3000.161} C_VEL
LIN {X 0,Y 559.674,Z 231.729,A -85,B 0,C 180,E1 -3002.717,E2 -3002.717} C_VEL
LIN {X 0,Y 559.818,Z 224.121,A -85,B 0,C 180,E1 -3005.311,E2 -3005.311} C_VEL
LIN {X 0,Y 559.183,Z 218.834,A -85,B 0,C 180,E1 -3007.275,E2 -3007.275} C_VEL
LIN {X 0,Y 559.165,Z 218.837,A -85,B 0,C 180,E1 -3009.941,E2 -3009.941} C_VEL
LIN {X 0,Y 559.163,Z 218.835,A -85,B 0,C 180,E1 -3012.742,E2 -3012.742} C_VEL
LIN {X 0,Y 559.148,Z 218.838,A -85,B 0,C 180,E1 -3015.76,E2 -3015.76} C_VEL
LIN {X 0,Y 559.191,Z 218.831,A -85,B 0,C 180,E1 -3018.232,E2 -3018.232} C_VEL
LIN {X 0,Y 559.174,Z 218.836,A -85,B 0,C 180,E1 -3021.191,E2 -3021.191} C_VEL
LIN {X 0,Y 559.157,Z 218.836,A -85,B 0,C 180,E1 -3023.79,E2 -3023.79} C_VEL
LIN {X 0,Y 559.163,Z 218.835,A -85,B 0,C 180,E1 -3026.424,E2 -3026.424} C_VEL
LIN {X 0,Y 559.151,Z 218.839,A -85,B 0,C 180,E1 -3028.98,E2 -3028.98} C_VEL
LIN {X 0,Y 559.168,Z 218.834,A -85,B 0,C 180,E1 -3031.617,E2 -3031.617} C_VEL
LIN {X 0,Y 559.179,Z 218.833,A -85,B 0,C 180,E1 -3033.902,E2 -3033.902} C_VEL
LIN {X 0,Y 559.136,Z 218.838,A -85,B 0,C 180,E1 -3036.571,E2 -3036.571} C_VEL
LIN {X 0,Y 559.177,Z 218.834,A -85,B 0,C 180,E1 -3039.394,E2 -3039.394} C_VEL
LIN {X 0,Y 559.145,Z 218.838,A -85,B 0,C 180,E1 -3041.685,E2 -3041.685} C_VEL
LIN {X 0,Y 559.165,Z 218.835,A -85,B 0,C 180,E1 -3043.947,E2 -3043.947} C_VEL
LIN {X 0,Y 559.171,Z 218.835,A -85,B 0,C 180,E1 -3046.183,E2 -3046.183} C_VEL
LIN {X 0,Y 559.191,Z 218.832,A -85,B 0,C 180,E1 -3049.132,E2 -3049.132} C_VEL
LIN {X 0,Y 559.203,Z 218.83,A -85,B 0,C 180,E1 -3052.053,E2 -3052.053} C_VEL
LIN {X 0,Y 559.251,Z 218.826,A -85,B 0,C 180,E1 -3054.952,E2 -3054.952} C_VEL
LIN {X 0,Y 559.243,Z 218.825,A -85,B 0,C 180,E1 -3057.838,E2 -3057.838} C_VEL
LIN {X 0,Y 559.273,Z 218.824,A -85,B 0,C 180,E1 -3060.719,E2 -3060.719} C_VEL
LIN {X 0,Y 559.238,Z 218.827,A -85,B 0,C 180,E1 -3062.88,E2 -3062.88} C_VEL
LIN {X 0,Y 559.224,Z 218.827,A -85,B 0,C 180,E1 -3065.769,E2 -3065.769} C_VEL
LIN {X 0,Y 559.197,Z 218.833,A -85,B 0,C 180,E1 -3068.673,E2 -3068.673} C_VEL
LIN {X 0,Y 559.202,Z 218.83,A -85,B 0,C 180,E1 -3071.599,E2 -3071.599} C_VEL
LIN {X 0,Y 559.19,Z 218.833,A -85,B 0,C 180,E1 -3074.594,E2 -3074.594} C_VEL
LIN {X 0,Y 559.113,Z 218.843,A -85,B 0,C 180,E1 -3077.557,E2 -3077.557} C_VEL
LIN {X 0,Y 559.009,Z 219.03,A -85,B 0,C 180,E1 -3079.078,E2 -3079.078} C_VEL
LIN {X 0,Y 558.953,Z 222.589,A -85,B 0,C 180,E1 -3082.159,E2 -3082.159} C_VEL
LIN {X 0,Y 558.952,Z 226.188,A -85,B 0,C 180,E1 -3085.307,E2 -3085.307} C_VEL
LIN {X 0,Y 558.892,Z 229.805,A -85,B 0,C 180,E1 -3088.33,E2 -3088.33} C_VEL
LIN {X 0,Y 558.847,Z 232.245,A -85,B 0,C 180,E1 -3090.511,E2 -3090.511} C_VEL
LIN {X 0,Y 558.164,Z 232.944,A -85,B 0,C 180,E1 -3091.108,E2 -3091.108} C_VEL
LIN {X 0,Y 555.27,Z 234.25,A -85,B 0,C 180,E1 -3092.075,E2 -3092.075} C_VEL
LIN {X 0,Y 552.834,Z 235.314,A -85,B 0,C 180,E1 -3092.853,E2 -3092.853} C_VEL
LIN {X 0,Y 551.795,Z 236.062,A -85,B 0,C 180,E1 -3093.455,E2 -3093.455} C_VEL
LIN {X 0,Y 551.714,Z 236.292,A -85,B 0,C 180,E1 -3093.659,E2 -3093.659} C_VEL
LIN {X 0,Y 551.64,Z 239.602,A -85,B 0,C 180,E1 -3096.619,E2 -3096.619} C_VEL
LIN {X 0,Y 551.633,Z 243.014,A -85,B 0,C 180,E1 -3099.568,E2 -3099.568} C_VEL
LIN {X 0,Y 551.667,Z 243.678,A -85,B 0,C 180,E1 -3100.099,E2 -3100.099} C_VEL
LIN {X 0,Y 553.015,Z 253.289,A -85,B 0,C 180,E1 -3100.364,E2 -3100.364} C_VEL
LIN {X 0,Y 552.894,Z 265.394,A -85,B 0,C 180,E1 -3100.769,E2 -3100.769} C_VEL
LIN {X 0,Y 552.645,Z 277.379,A -85,B 0,C 180,E1 -3101.316,E2 -3101.316} C_VEL
LIN {X 0,Y 552.489,Z 289.217,A -85,B 0,C 180,E1 -3102.02,E2 -3102.02} C_VEL
LIN {X 0,Y 552.331,Z 299.297,A -85,B 0,C 180,E1 -3102.775,E2 -3102.775} C_VEL
LIN {X 0,Y 552.146,Z 309.198,A -85,B 0,C 180,E1 -3103.691,E2 -3103.691} C_VEL
LIN {X 0,Y 551.981,Z 318.705,A -85,B 0,C 180,E1 -3104.778,E2 -3104.778} C_VEL
LIN {X 0,Y 551.912,Z 325.931,A -85,B 0,C 180,E1 -3105.8,E2 -3105.8} C_VEL
LIN {X 0,Y 551.801,Z 332.944,A -85,B 0,C 180,E1 -3107.048,E2 -3107.048} C_VEL
LIN {X 0,Y 551.769,Z 337.516,A -85,B 0,C 180,E1 -3108.076,E2 -3108.076} C_VEL
LIN {X 0,Y 551.73,Z 341.109,A -85,B 0,C 180,E1 -3109.101,E2 -3109.101} C_VEL
LIN {X 0,Y 551.661,Z 344.431,A -85,B 0,C 180,E1 -3110.434,E2 -3110.434} C_VEL
LIN {X 0,Y 551.634,Z 345.951,A -85,B 0,C 180,E1 -3111.372,E2 -3111.372} C_VEL
LIN {X 0,Y 551.65,Z 346.778,A -85,B 0,C 180,E1 -3112.302,E2 -3112.302} C_VEL
LIN {X 0,Y 551.64,Z 346.934,A -85,B 0,C 180,E1 -3113.379,E2 -3113.379} C_VEL
LIN {X 0,Y 551.66,Z 346.059,A -85,B 0,C 180,E1 -3114.618,E2 -3114.618} C_VEL
LIN {X 0,Y 551.697,Z 343.925,A -85,B 0,C 180,E1 -3115.91,E2 -3115.91} C_VEL
LIN {X 0,Y 551.704,Z 340.394,A -85,B 0,C 180,E1 -3117.217,E2 -3117.217} C_VEL
LIN {X 0,Y 551.779,Z 335.142,A -85,B 0,C 180,E1 -3118.578,E2 -3118.578} C_VEL
LIN {X 0,Y 551.868,Z 329.381,A -85,B 0,C 180,E1 -3119.715,E2 -3119.715} C_VEL
LIN {X 0,Y 551.962,Z 322.105,A -85,B 0,C 180,E1 -3120.855,E2 -3120.855} C_VEL
LIN {X 0,Y 552.042,Z 313.828,A -85,B 0,C 180,E1 -3121.899,E2 -3121.899} C_VEL
LIN {X 0,Y 552.23,Z 304.184,A -85,B 0,C 180,E1 -3122.887,E2 -3122.887} C_VEL
LIN {X 0,Y 552.434,Z 293.539,A -85,B 0,C 180,E1 -3123.764,E2 -3123.764} C_VEL
LIN {X 0,Y 552.612,Z 281.539,A -85,B 0,C 180,E1 -3124.546,E2 -3124.546} C_VEL
LIN {X 0,Y 552.796,Z 269.615,A -85,B 0,C 180,E1 -3125.149,E2 -3125.149} C_VEL
LIN {X 0,Y 552.972,Z 256.564,A -85,B 0,C 180,E1 -3125.629,E2 -3125.629} C_VEL
LIN {X 0,Y 552.74,Z 249.977,A -85,B 0,C 180,E1 -3125.818,E2 -3125.818} C_VEL
LIN {X 0,Y 551.672,Z 243.688,A -85,B 0,C 180,E1 -3125.983,E2 -3125.983} C_VEL
LIN {X 0,Y 551.687,Z 239.931,A -85,B 0,C 180,E1 -3129.103,E2 -3129.103} C_VEL
LIN {X 0,Y 551.697,Z 237.229,A -85,B 0,C 180,E1 -3131.43,E2 -3131.43} C_VEL
LIN {X 0,Y 551.735,Z 234.628,A -85,B 0,C 180,E1 -3133.727,E2 -3133.727} C_VEL
LIN {X 0,Y 551.81,Z 231.991,A -85,B 0,C 180,E1 -3135.997,E2 -3135.997} C_VEL
LIN {X 0,Y 551.856,Z 228.535,A -85,B 0,C 180,E1 -3138.988,E2 -3138.988} C_VEL
LIN {X 0,Y 551.88,Z 225.125,A -85,B 0,C 180,E1 -3141.948,E2 -3141.948} C_VEL
LIN {X 0,Y 551.93,Z 221.771,A -85,B 0,C 180,E1 -3144.887,E2 -3144.887} C_VEL
LIN {X 0,Y 551.874,Z 220.089,A -85,B 0,C 180,E1 -3146.35,E2 -3146.35} C_VEL
LIN {X 0,Y 552.137,Z 219.713,A -85,B 0,C 180,E1 -3147.812,E2 -3147.812} C_VEL
LIN {X 0,Y 552.216,Z 219.7,A -85,B 0,C 180,E1 -3150.001,E2 -3150.001} C_VEL
LIN {X 0,Y 552.195,Z 219.705,A -85,B 0,C 180,E1 -3152.919,E2 -3152.919} C_VEL
LIN {X 0,Y 552.189,Z 219.703,A -85,B 0,C 180,E1 -3155.845,E2 -3155.845} C_VEL
LIN {X 0,Y 552.161,Z 219.709,A -85,B 0,C 180,E1 -3158.786,E2 -3158.786} C_VEL
LIN {X 0,Y 552.152,Z 219.709,A -85,B 0,C 180,E1 -3161.751,E2 -3161.751} C_VEL
LIN {X 0,Y 552.124,Z 219.712,A -85,B 0,C 180,E1 -3164.749,E2 -3164.749} C_VEL
LIN {X 0,Y 552.104,Z 219.716,A -85,B 0,C 180,E1 -3167.789,E2 -3167.789} C_VEL
LIN {X 0,Y 552.123,Z 219.713,A -85,B 0,C 180,E1 -3170.102,E2 -3170.102} C_VEL
LIN {X 0,Y 552.103,Z 219.716,A -85,B 0,C 180,E1 -3172.451,E2 -3172.451} C_VEL
LIN {X 0,Y 552.146,Z 219.709,A -85,B 0,C 180,E1 -3175.352,E2 -3175.352} C_VEL
LIN {X 0,Y 552.118,Z 219.714,A -85,B 0,C 180,E1 -3178.099,E2 -3178.099} C_VEL
LIN {X 0,Y 552.098,Z 219.716,A -85,B 0,C 180,E1 -3180.61,E2 -3180.61} C_VEL
LIN {X 0,Y 552.121,Z 219.712,A -85,B 0,C 180,E1 -3183.186,E2 -3183.186} C_VEL
LIN {X 0,Y 552.106,Z 219.714,A -85,B 0,C 180,E1 -3185.843,E2 -3185.843} C_VEL
LIN {X 0,Y 552.118,Z 219.712,A -85,B 0,C 180,E1 -3189.063,E2 -3189.063} C_VEL
LIN {X 0,Y 552.134,Z 219.71,A -85,B 0,C 180,E1 -3191.446,E2 -3191.446} C_VEL
LIN {X 0,Y 552.091,Z 219.716,A -85,B 0,C 180,E1 -3194.534,E2 -3194.534} C_VEL
LIN {X 0,Y 552.126,Z 219.713,A -85,B 0,C 180,E1 -3197.586,E2 -3197.586} C_VEL
LIN {X 0,Y 552.131,Z 219.711,A -85,B 0,C 180,E1 -3200.475,E2 -3200.475} C_VEL
LIN {X 0,Y 552.111,Z 219.715,A -85,B 0,C 180,E1 -3203.317,E2 -3203.317} C_VEL
LIN {X 0,Y 552.126,Z 219.711,A -85,B 0,C 180,E1 -3205.941,E2 -3205.941} C_VEL
LIN {X 0,Y 552.118,Z 219.713,A -85,B 0,C 180,E1 -3208.542,E2 -3208.542} C_VEL
LIN {X 0,Y 552.124,Z 219.713,A -85,B 0,C 180,E1 -3211.44,E2 -3211.44} C_VEL
LIN {X 0,Y 552.131,Z 219.711,A -85,B 0,C 180,E1 -3214.357,E2 -3214.357} C_VEL
LIN {X 0,Y 552.097,Z 219.716,A -85,B 0,C 180,E1 -3216.759,E2 -3216.759} C_VEL
LIN {X 0,Y 552.123,Z 219.713,A -85,B 0,C 180,E1 -3219.121,E2 -3219.121} C_VEL
LIN {X 0,Y 552.126,Z 219.712,A -85,B 0,C 180,E1 -3221.446,E2 -3221.446} C_VEL
LIN {X 0,Y 552.115,Z 219.714,A -85,B 0,C 180,E1 -3223.739,E2 -3223.739} C_VEL
LIN {X 0,Y 552.139,Z 219.711,A -85,B 0,C 180,E1 -3226.006,E2 -3226.006} C_VEL
LIN {X 0,Y 552.165,Z 219.705,A -85,B 0,C 180,E1 -3228.995,E2 -3228.995} C_VEL
LIN {X 0,Y 552.152,Z 219.71,A -85,B 0,C 180,E1 -3231.953,E2 -3231.953} C_VEL
LIN {X 0,Y 552.231,Z 219.698,A -85,B 0,C 180,E1 -3234.89,E2 -3234.89} C_VEL
LIN {X 0,Y 552.221,Z 219.7,A -85,B 0,C 180,E1 -3237.813,E2 -3237.813} C_VEL
LIN {X 0,Y 552.244,Z 219.697,A -85,B 0,C 180,E1 -3240.73,E2 -3240.73} C_VEL
LIN {X 0,Y 552.206,Z 219.7,A -85,B 0,C 180,E1 -3242.919,E2 -3242.919} C_VEL
LIN {X 0,Y 552.199,Z 219.703,A -85,B 0,C 180,E1 -3245.845,E2 -3245.845} C_VEL
LIN {X 0,Y 552.148,Z 219.709,A -85,B 0,C 180,E1 -3248.787,E2 -3248.787} C_VEL
LIN {X 0,Y 552.17,Z 219.706,A -85,B 0,C 180,E1 -3251.751,E2 -3251.751} C_VEL
LIN {X 0,Y 552.138,Z 219.712,A -85,B 0,C 180,E1 -3254.749,E2 -3254.749} C_VEL
LIN {X 0,Y 552.102,Z 219.715,A -85,B 0,C 180,E1 -3257.79,E2 -3257.79} C_VEL
LIN {X 0,Y 552.135,Z 219.71,A -85,B 0,C 180,E1 -3260.102,E2 -3260.102} C_VEL
LIN {X 0,Y 552.099,Z 219.715,A -85,B 0,C 180,E1 -3262.452,E2 -3262.452} C_VEL
LIN {X 0,Y 552.117,Z 219.712,A -85,B 0,C 180,E1 -3265.646,E2 -3265.646} C_VEL
LIN {X 0,Y 552.133,Z 219.713,A -85,B 0,C 180,E1 -3268.562,E2 -3268.562} C_VEL
LIN {X 0,Y 552.121,Z 219.712,A -85,B 0,C 180,E1 -3271.476,E2 -3271.476} C_VEL
LIN {X 0,Y 552.133,Z 219.712,A -85,B 0,C 180,E1 -3274.169,E2 -3274.169} C_VEL
LIN {X 0,Y 552.114,Z 219.714,A -85,B 0,C 180,E1 -3276.747,E2 -3276.747} C_VEL
LIN {X 0,Y 552.137,Z 219.71,A -85,B 0,C 180,E1 -3279.527,E2 -3279.527} C_VEL
LIN {X 0,Y 552.138,Z 219.711,A -85,B 0,C 180,E1 -3282.425,E2 -3282.425} C_VEL
LIN {X 0,Y 552.1,Z 219.716,A -85,B 0,C 180,E1 -3285.562,E2 -3285.562} C_VEL
LIN {X 0,Y 552.129,Z 219.71,A -85,B 0,C 180,E1 -3288.554,E2 -3288.554} C_VEL
LIN {X 0,Y 552.123,Z 219.714,A -85,B 0,C 180,E1 -3291.411,E2 -3291.411} C_VEL
LIN {X 0,Y 552.136,Z 219.816,A -85,B 0,C 180,E1 -3292.569,E2 -3292.569} C_VEL
LIN {X 0,Y 552.853,Z 224.942,A -85,B 0,C 180,E1 -3294.448,E2 -3294.448} C_VEL
LIN {X 0,Y 552.745,Z 232.558,A -85,B 0,C 180,E1 -3297.054,E2 -3297.054} C_VEL
LIN {X 0,Y 552.557,Z 239.744,A -85,B 0,C 180,E1 -3299.418,E2 -3299.418} C_VEL
LIN {X 0,Y 552.432,Z 247.757,A -85,B 0,C 180,E1 -3301.919,E2 -3301.919} C_VEL
LIN {X 0,Y 552.336,Z 256.587,A -85,B 0,C 180,E1 -3304.611,E2 -3304.611} C_VEL
LIN {X 0,Y 552.165,Z 266.35,A -85,B 0,C 180,E1 -3307.551,E2 -3307.551} C_VEL
LIN {X 0,Y 552.085,Z 276.153,A -85,B 0,C 180,E1 -3310.394,E2 -3310.394} C_VEL
LIN {X 0,Y 551.998,Z 286.691,A -85,B 0,C 180,E1 -3313.353,E2 -3313.353} C_VEL
LIN {X 0,Y 551.917,Z 297.376,A -85,B 0,C 180,E1 -3316.374,E2 -3316.374} C_VEL
LIN {X 0,Y 551.888,Z 299.528,A -85,B 0,C 180,E1 -3316.982,E2 -3316.982} C_VEL
LIN {X 0,Y 553.102,Z 308.491,A -85,B 0,C 180,E1 -3317.198,E2 -3317.198} C_VEL
LIN {X 0,Y 552.922,Z 321.154,A -85,B 0,C 180,E1 -3317.567,E2 -3317.567} C_VEL
LIN {X 0,Y 552.747,Z 333.475,A -85,B 0,C 180,E1 -3318.075,E2 -3318.075} C_VEL
LIN {X 0,Y 552.579,Z 345.219,A -85,B 0,C 180,E1 -3318.717,E2 -3318.717} C_VEL
LIN {X 0,Y 552.427,Z 357.084,A -85,B 0,C 180,E1 -3319.554,E2 -3319.554} C_VEL
LIN {X 0,Y 552.202,Z 367.532,A -85,B 0,C 180,E1 -3320.476,E2 -3320.476} C_VEL
LIN {X 0,Y 552.079,Z 375.986,A -85,B 0,C 180,E1 -3321.397,E2 -3321.397} C_VEL
LIN {X 0,Y 551.928,Z 384.231,A -85,B 0,C 180,E1 -3322.5,E2 -3322.5} C_VEL
LIN {X 0,Y 551.823,Z 391.208,A -85,B 0,C 180,E1 -3323.662,E2 -3323.662} C_VEL
LIN {X 0,Y 551.724,Z 396.947,A -85,B 0,C 180,E1 -3324.884,E2 -3324.884} C_VEL
LIN {X 0,Y 551.764,Z 400.892,A -85,B 0,C 180,E1 -3325.982,E2 -3325.982} C_VEL
LIN {X 0,Y 551.724,Z 403.806,A -85,B 0,C 180,E1 -3327.079,E2 -3327.079} C_VEL
LIN {X 0,Y 551.645,Z 406.183,A -85,B 0,C 180,E1 -3328.539,E2 -3328.539} C_VEL
LIN {X 0,Y 551.64,Z 407,A -85,B 0,C 180,E1 -3329.999,E2 -3329.999} C_VEL
LIN {X 0,Y 551.645,Z 406.185,A -85,B 0,C 180,E1 -3331.459,E2 -3331.459} C_VEL
LIN {X 0,Y 551.724,Z 403.812,A -85,B 0,C 180,E1 -3332.92,E2 -3332.92} C_VEL
LIN {X 0,Y 551.764,Z 400.898,A -85,B 0,C 180,E1 -3334.016,E2 -3334.016} C_VEL
LIN {X 0,Y 551.724,Z 396.951,A -85,B 0,C 180,E1 -3335.115,E2 -3335.115} C_VEL
LIN {X 0,Y 551.814,Z 391.135,A -85,B 0,C 180,E1 -3336.351,E2 -3336.351} C_VEL
LIN {X 0,Y 551.926,Z 384.241,A -85,B 0,C 180,E1 -3337.499,E2 -3337.499} C_VEL
LIN {X 0,Y 552.082,Z 375.998,A -85,B 0,C 180,E1 -3338.602,E2 -3338.602} C_VEL
LIN {X 0,Y 552.201,Z 367.547,A -85,B 0,C 180,E1 -3339.523,E2 -3339.523} C_VEL
LIN {X 0,Y 552.426,Z 357.103,A -85,B 0,C 180,E1 -3340.444,E2 -3340.444} C_VEL
LIN {X 0,Y 552.593,Z 345.291,A -85,B 0,C 180,E1 -3341.279,E2 -3341.279} C_VEL
LIN {X 0,Y 552.742,Z 333.504,A -85,B 0,C 180,E1 -3341.923,E2 -3341.923} C_VEL
LIN {X 0,Y 552.954,Z 321.187,A -85,B 0,C 180,E1 -3342.431,E2 -3342.431} C_VEL
LIN {X 0,Y 553.079,Z 308.546,A -85,B 0,C 180,E1 -3342.801,E2 -3342.801} C_VEL
LIN {X 0,Y 552.263,Z 302.029,A -85,B 0,C 180,E1 -3342.955,E2 -3342.955} C_VEL
LIN {X 0,Y 551.887,Z 299.533,A -85,B 0,C 180,E1 -3343.016,E2 -3343.016} C_VEL
LIN {X 0,Y 551.974,Z 289.417,A -85,B 0,C 180,E1 -3345.887,E2 -3345.887} C_VEL
LIN {X 0,Y 552.087,Z 278.437,A -85,B 0,C 180,E1 -3348.941,E2 -3348.941} C_VEL
LIN {X 0,Y 552.175,Z 267.38,A -85,B 0,C 180,E1 -3352.052,E2 -3352.052} C_VEL
LIN {X 0,Y 552.2,Z 257.787,A -85,B 0,C 180,E1 -3354.834,E2 -3354.834} C_VEL
LIN {X 0,Y 552.322,Z 248.692,A -85,B 0,C 180,E1 -3357.673,E2 -3357.673} C_VEL
LIN {X 0,Y 552.518,Z 240.903,A -85,B 0,C 180,E1 -3360.121,E2 -3360.121} C_VEL
LIN {X 0,Y 552.706,Z 232.36,A -85,B 0,C 180,E1 -3362.94,E2 -3362.94} C_VEL
LIN {X 0,Y 552.843,Z 224.873,A -85,B 0,C 180,E1 -3365.55,E2 -3365.55} C_VEL
LIN {X 0,Y 552.112,Z 219.716,A -85,B 0,C 180,E1 -3367.546,E2 -3367.546} C_VEL
LIN {X 0,Y 552.121,Z 219.713,A -85,B 0,C 180,E1 -3370.479,E2 -3370.479} C_VEL
LIN {X 0,Y 552.104,Z 219.715,A -85,B 0,C 180,E1 -3373.482,E2 -3373.482} C_VEL
LIN {X 0,Y 552.105,Z 219.717,A -85,B 0,C 180,E1 -3376.575,E2 -3376.575} C_VEL
LIN {X 0,Y 552.12,Z 219.712,A -85,B 0,C 180,E1 -3379.519,E2 -3379.519} C_VEL
LIN {X 0,Y 552.091,Z 219.718,A -85,B 0,C 180,E1 -3382.335,E2 -3382.335} C_VEL
LIN {X 0,Y 552.124,Z 219.712,A -85,B 0,C 180,E1 -3385.053,E2 -3385.053} C_VEL
LIN {X 0,Y 552.123,Z 219.713,A -85,B 0,C 180,E1 -3387.681,E2 -3387.681} C_VEL
LIN {X 0,Y 552.109,Z 219.716,A -85,B 0,C 180,E1 -3390.234,E2 -3390.234} C_VEL
LIN {X 0,Y 552.139,Z 219.71,A -85,B 0,C 180,E1 -3392.998,E2 -3392.998} C_VEL
LIN {X 0,Y 552.11,Z 219.713,A -85,B 0,C 180,E1 -3395.16,E2 -3395.16} C_VEL
LIN {X 0,Y 552.122,Z 219.712,A -85,B 0,C 180,E1 -3398.336,E2 -3398.336} C_VEL
LIN {X 0,Y 552.153,Z 219.708,A -85,B 0,C 180,E1 -3400.673,E2 -3400.673} C_VEL
LIN {X 0,Y 552.115,Z 219.715,A -85,B 0,C 180,E1 -3403.736,E2 -3403.736} C_VEL
LIN {X 0,Y 552.134,Z 219.713,A -85,B 0,C 180,E1 -3406.003,E2 -3406.003} C_VEL
LIN {X 0,Y 552.158,Z 219.707,A -85,B 0,C 180,E1 -3408.992,E2 -3408.992} C_VEL
LIN {X 0,Y 552.157,Z 219.708,A -85,B 0,C 180,E1 -3411.95,E2 -3411.95} C_VEL
LIN {X 0,Y 552.226,Z 219.7,A -85,B 0,C 180,E1 -3414.888,E2 -3414.888} C_VEL
LIN {X 0,Y 552.215,Z 219.7,A -85,B 0,C 180,E1 -3417.811,E2 -3417.811} C_VEL
LIN {X 0,Y 552.242,Z 219.7,A -85,B 0,C 180,E1 -3420.728,E2 -3420.728} C_VEL
LIN {X 0,Y 552.204,Z 219.704,A -85,B 0,C 180,E1 -3422.917,E2 -3422.917} C_VEL
LIN {X 0,Y 552.194,Z 219.703,A -85,B 0,C 180,E1 -3425.843,E2 -3425.843} C_VEL
LIN {X 0,Y 552.165,Z 219.708,A -85,B 0,C 180,E1 -3428.784,E2 -3428.784} C_VEL
LIN {X 0,Y 552.157,Z 219.708,A -85,B 0,C 180,E1 -3431.749,E2 -3431.749} C_VEL
LIN {X 0,Y 552.128,Z 219.712,A -85,B 0,C 180,E1 -3434.747,E2 -3434.747} C_VEL
LIN {X 0,Y 552.099,Z 219.716,A -85,B 0,C 180,E1 -3437.311,E2 -3437.311} C_VEL
LIN {X 0,Y 551.995,Z 219.731,A -85,B 0,C 180,E1 -3438.559,E2 -3438.559} C_VEL
LIN {X 0,Y 551.913,Z 220.291,A -85,B 0,C 180,E1 -3439.56,E2 -3439.56} C_VEL
LIN {X 0,Y 551.894,Z 223.621,A -85,B 0,C 180,E1 -3442.458,E2 -3442.458} C_VEL
LIN {X 0,Y 551.864,Z 227.229,A -85,B 0,C 180,E1 -3445.656,E2 -3445.656} C_VEL
LIN {X 0,Y 551.804,Z 230.577,A -85,B 0,C 180,E1 -3448.502,E2 -3448.502} C_VEL
LIN {X 0,Y 551.801,Z 233.035,A -85,B 0,C 180,E1 -3450.626,E2 -3450.626} C_VEL
LIN {X 0,Y 551.714,Z 236.292,A -85,B 0,C 180,E1 -3453.659,E2 -3453.659} C_VEL
LIN {X 0,Y 551.041,Z 237.016,A -85,B 0,C 180,E1 -3454.264,E2 -3454.264} C_VEL
LIN {X 0,Y 548.128,Z 238.351,A -85,B 0,C 180,E1 -3455.242,E2 -3455.242} C_VEL
LIN {X 0,Y 545.679,Z 239.437,A -85,B 0,C 180,E1 -3456.03,E2 -3456.03} C_VEL
LIN {X 0,Y 544.651,Z 240.205,A -85,B 0,C 180,E1 -3456.64,E2 -3456.64} C_VEL
LIN {X 0,Y 544.581,Z 240.443,A -85,B 0,C 180,E1 -3456.846,E2 -3456.846} C_VEL
LIN {X 0,Y 544.579,Z 243.983,A -85,B 0,C 180,E1 -3459.935,E2 -3459.935} C_VEL
LIN {X 0,Y 546.116,Z 253.853,A -85,B 0,C 180,E1 -3460.211,E2 -3460.211} C_VEL
LIN {X 0,Y 545.944,Z 266.73,A -85,B 0,C 180,E1 -3460.659,E2 -3460.659} C_VEL
LIN {X 0,Y 545.668,Z 278.7,A -85,B 0,C 180,E1 -3461.227,E2 -3461.227} C_VEL
LIN {X 0,Y 545.485,Z 290.109,A -85,B 0,C 180,E1 -3461.933,E2 -3461.933} C_VEL
LIN {X 0,Y 545.3,Z 300.262,A -85,B 0,C 180,E1 -3462.725,E2 -3462.725} C_VEL
LIN {X 0,Y 545.118,Z 309.567,A -85,B 0,C 180,E1 -3463.608,E2 -3463.608} C_VEL
LIN {X 0,Y 544.946,Z 318.525,A -85,B 0,C 180,E1 -3464.648,E2 -3464.648} C_VEL
LIN {X 0,Y 544.856,Z 325.793,A -85,B 0,C 180,E1 -3465.684,E2 -3465.684} C_VEL
LIN {X 0,Y 544.738,Z 332.415,A -85,B 0,C 180,E1 -3466.861,E2 -3466.861} C_VEL
LIN {X 0,Y 544.673,Z 338.159,A -85,B 0,C 180,E1 -3468.179,E2 -3468.179} C_VEL
LIN {X 0,Y 544.628,Z 341.657,A -85,B 0,C 180,E1 -3469.24,E2 -3469.24} C_VEL
LIN {X 0,Y 544.624,Z 343.174,A -85,B 0,C 180,E1 -3469.819,E2 -3469.819} C_VEL
LIN {X 0,Y 544.551,Z 345.117,A -85,B 0,C 180,E1 -3470.774,E2 -3470.774} C_VEL
LIN {X 0,Y 544.529,Z 346.543,A -85,B 0,C 180,E1 -3471.931,E2 -3471.931} C_VEL
LIN {X 0,Y 544.554,Z 346.985,A -85,B 0,C 180,E1 -3473.143,E2 -3473.143} C_VEL
LIN {X 0,Y 544.549,Z 346.213,A -85,B 0,C 180,E1 -3474.496,E2 -3474.496} C_VEL
LIN {X 0,Y 544.573,Z 344.444,A -85,B 0,C 180,E1 -3475.682,E2 -3475.682} C_VEL
LIN {X 0,Y 544.599,Z 341.189,A -85,B 0,C 180,E1 -3477.012,E2 -3477.012} C_VEL
LIN {X 0,Y 544.682,Z 336.306,A -85,B 0,C 180,E1 -3478.382,E2 -3478.382} C_VEL
LIN {X 0,Y 544.776,Z 330.586,A -85,B 0,C 180,E1 -3479.58,E2 -3479.58} C_VEL
LIN {X 0,Y 544.887,Z 323.027,A -85,B 0,C 180,E1 -3480.825,E2 -3480.825} C_VEL
LIN {X 0,Y 545.012,Z 314.619,A -85,B 0,C 180,E1 -3481.923,E2 -3481.923} C_VEL
LIN {X 0,Y 545.201,Z 305.137,A -85,B 0,C 180,E1 -3482.924,E2 -3482.924} C_VEL
LIN {X 0,Y 545.434,Z 294.782,A -85,B 0,C 180,E1 -3483.813,E2 -3483.813} C_VEL
LIN {X 0,Y 545.59,Z 283.967,A -85,B 0,C 180,E1 -3484.557,E2 -3484.557} C_VEL
LIN {X 0,Y 545.803,Z 271.772,A -85,B 0,C 180,E1 -3485.211,E2 -3485.211} C_VEL
LIN {X 0,Y 546.022,Z 260.218,A -85,B 0,C 180,E1 -3485.678,E2 -3485.678} C_VEL
LIN {X 0,Y 545.912,Z 251.326,A -85,B 0,C 180,E1 -3485.95,E2 -3485.95} C_VEL
LIN {X 0,Y 544.594,Z 243.919,A -85,B 0,C 180,E1 -3486.154,E2 -3486.154} C_VEL
LIN {X 0,Y 544.614,Z 240.759,A -85,B 0,C 180,E1 -3488.819,E2 -3488.819} C_VEL
LIN {X 0,Y 544.639,Z 238.044,A -85,B 0,C 180,E1 -3491.181,E2 -3491.181} C_VEL
LIN {X 0,Y 544.685,Z 235.432,A -85,B 0,C 180,E1 -3493.51,E2 -3493.51} C_VEL
LIN {X 0,Y 544.742,Z 232.796,A -85,B 0,C 180,E1 -3495.811,E2 -3495.811} C_VEL
LIN {X 0,Y 544.809,Z 229.284,A -85,B 0,C 180,E1 -3498.844,E2 -3498.844} C_VEL
LIN {X 0,Y 544.809,Z 225.893,A -85,B 0,C 180,E1 -3501.843,E2 -3501.843} C_VEL
LIN {X 0,Y 544.795,Z 223.349,A -85,B 0,C 180,E1 -3504.077,E2 -3504.077} C_VEL
LIN {X 0,Y 544.816,Z 220.8,A -85,B 0,C 180,E1 -3506.303,E2 -3506.303} C_VEL
LIN {X 0,Y 545.101,Z 220.589,A -85,B 0,C 180,E1 -3507.784,E2 -3507.784} C_VEL
LIN {X 0,Y 545.186,Z 220.575,A -85,B 0,C 180,E1 -3510.001,E2 -3510.001} C_VEL
LIN {X 0,Y 545.162,Z 220.581,A -85,B 0,C 180,E1 -3512.957,E2 -3512.957} C_VEL
LIN {X 0,Y 545.16,Z 220.579,A -85,B 0,C 180,E1 -3515.92,E2 -3515.92} C_VEL
LIN {X 0,Y 545.117,Z 220.585,A -85,B 0,C 180,E1 -3518.901,E2 -3518.901} C_VEL
LIN {X 0,Y 545.123,Z 220.585,A -85,B 0,C 180,E1 -3521.905,E2 -3521.905} C_VEL
LIN {X 0,Y 545.073,Z 220.59,A -85,B 0,C 180,E1 -3524.945,E2 -3524.945} C_VEL
LIN {X 0,Y 545.072,Z 220.59,A -85,B 0,C 180,E1 -3528.027,E2 -3528.027} C_VEL
LIN {X 0,Y 545.088,Z 220.589,A -85,B 0,C 180,E1 -3530.373,E2 -3530.373} C_VEL
LIN {X 0,Y 545.103,Z 220.587,A -85,B 0,C 180,E1 -3533.559,E2 -3533.559} C_VEL
LIN {X 0,Y 545.079,Z 220.59,A -85,B 0,C 180,E1 -3536.001,E2 -3536.001} C_VEL
LIN {X 0,Y 545.081,Z 220.589,A -85,B 0,C 180,E1 -3538.75,E2 -3538.75} C_VEL
LIN {X 0,Y 545.069,Z 220.591,A -85,B 0,C 180,E1 -3541.684,E2 -3541.684} C_VEL
LIN {X 0,Y 545.077,Z 220.59,A -85,B 0,C 180,E1 -3544.564,E2 -3544.564} C_VEL
LIN {X 0,Y 545.032,Z 220.596,A -85,B 0,C 180,E1 -3547.305,E2 -3547.305} C_VEL
LIN {X 0,Y 545.086,Z 220.588,A -85,B 0,C 180,E1 -3550.142,E2 -3550.142} C_VEL
LIN {X 0,Y 545.082,Z 220.589,A -85,B 0,C 180,E1 -3553.107,E2 -3553.107} C_VEL
LIN {X 0,Y 545.061,Z 220.592,A -85,B 0,C 180,E1 -3556.226,E2 -3556.226} C_VEL
LIN {X 0,Y 545.097,Z 220.587,A -85,B 0,C 180,E1 -3558.889,E2 -3558.889} C_VEL
LIN {X 0,Y 545.051,Z 220.592,A -85,B 0,C 180,E1 -3561.765,E2 -3561.765} C_VEL
LIN {X 0,Y 545.055,Z 220.594,A -85,B 0,C 180,E1 -3564.535,E2 -3564.535} C_VEL
LIN {X 0,Y 545.079,Z 220.588,A -85,B 0,C 180,E1 -3567.214,E2 -3567.214} C_VEL
LIN {X 0,Y 545.063,Z 220.591,A -85,B 0,C 180,E1 -3569.812,E2 -3569.812} C_VEL
LIN {X 0,Y 545.089,Z 220.59,A -85,B 0,C 180,E1 -3572.346,E2 -3572.346} C_VEL
LIN {X 0,Y 545.118,Z 220.585,A -85,B 0,C 180,E1 -3574.822,E2 -3574.822} C_VEL
LIN {X 0,Y 545.038,Z 220.595,A -85,B 0,C 180,E1 -3577.244,E2 -3577.244} C_VEL
LIN {X 0,Y 545.123,Z 220.586,A -85,B 0,C 180,E1 -3580.417,E2 -3580.417} C_VEL
LIN {X 0,Y 545.067,Z 220.59,A -85,B 0,C 180,E1 -3583.522,E2 -3583.522} C_VEL
LIN {X 0,Y 545.099,Z 220.587,A -85,B 0,C 180,E1 -3585.821,E2 -3585.821} C_VEL
LIN {X 0,Y 545.121,Z 220.583,A -85,B 0,C 180,E1 -3588.851,E2 -3588.851} C_VEL
LIN {X 0,Y 545.101,Z 220.589,A -85,B 0,C 180,E1 -3591.848,E2 -3591.848} C_VEL
LIN {X 0,Y 545.207,Z 220.572,A -85,B 0,C 180,E1 -3594.824,E2 -3594.824} C_VEL
LIN {X 0,Y 545.194,Z 220.576,A -85,B 0,C 180,E1 -3597.785,E2 -3597.785} C_VEL
LIN {X 0,Y 545.215,Z 220.572,A -85,B 0,C 180,E1 -3600.74,E2 -3600.74} C_VEL
LIN {X 0,Y 545.173,Z 220.577,A -85,B 0,C 180,E1 -3602.957,E2 -3602.957} C_VEL
LIN {X 0,Y 545.171,Z 220.578,A -85,B 0,C 180,E1 -3605.921,E2 -3605.921} C_VEL
LIN {X 0,Y 545.108,Z 220.586,A -85,B 0,C 180,E1 -3608.901,E2 -3608.901} C_VEL
LIN {X 0,Y 545.113,Z 220.585,A -85,B 0,C 180,E1 -3611.906,E2 -3611.906} C_VEL
LIN {X 0,Y 545.091,Z 220.589,A -85,B 0,C 180,E1 -3614.944,E2 -3614.944} C_VEL
LIN {X 0,Y 545.068,Z 220.592,A -85,B 0,C 180,E1 -3618.027,E2 -3618.027} C_VEL
LIN {X 0,Y 545.101,Z 220.588,A -85,B 0,C 180,E1 -3620.373,E2 -3620.373} C_VEL
LIN {X 0,Y 545.082,Z 220.589,A -85,B 0,C 180,E1 -3623.56,E2 -3623.56} C_VEL
LIN {X 0,Y 545.076,Z 220.591,A -85,B 0,C 180,E1 -3626.002,E2 -3626.002} C_VEL
LIN {X 0,Y 545.098,Z 220.588,A -85,B 0,C 180,E1 -3628.748,E2 -3628.748} C_VEL
LIN {X 0,Y 545.063,Z 220.593,A -85,B 0,C 180,E1 -3631.915,E2 -3631.915} C_VEL
LIN {X 0,Y 545.067,Z 220.591,A -85,B 0,C 180,E1 -3634.565,E2 -3634.565} C_VEL
LIN {X 0,Y 545.044,Z 220.594,A -85,B 0,C 180,E1 -3637.304,E2 -3637.304} C_VEL
LIN {X 0,Y 545.073,Z 220.591,A -85,B 0,C 180,E1 -3640.143,E2 -3640.143} C_VEL
LIN {X 0,Y 545.087,Z 220.589,A -85,B 0,C 180,E1 -3643.107,E2 -3643.107} C_VEL
LIN {X 0,Y 545.057,Z 220.59,A -85,B 0,C 180,E1 -3646.226,E2 -3646.226} C_VEL
LIN {X 0,Y 545.09,Z 220.588,A -85,B 0,C 180,E1 -3648.885,E2 -3648.885} C_VEL
LIN {X 0,Y 545.087,Z 220.589,A -85,B 0,C 180,E1 -3650.818,E2 -3650.818} C_VEL
LIN {X 0,Y 545.097,Z 220.731,A -85,B 0,C 180,E1 -3652.351,E2 -3652.351} C_VEL
LIN {X 0,Y 545.894,Z 225.688,A -85,B 0,C 180,E1 -3654.202,E2 -3654.202} C_VEL
LIN {X 0,Y 545.783,Z 233.213,A -85,B 0,C 180,E1 -3656.825,E2 -3656.825} C_VEL
LIN {X 0,Y 545.574,Z 240.853,A -85,B 0,C 180,E1 -3659.369,E2 -3659.369} C_VEL
LIN {X 0,Y 545.421,Z 248.917,A -85,B 0,C 180,E1 -3661.944,E2 -3661.944} C_VEL
LIN {X 0,Y 545.274,Z 258.206,A -85,B 0,C 180,E1 -3664.827,E2 -3664.827} C_VEL
LIN {X 0,Y 545.12,Z 267.451,A -85,B 0,C 180,E1 -3667.645,E2 -3667.645} C_VEL
LIN {X 0,Y 545.023,Z 276.862,A -85,B 0,C 180,E1 -3670.411,E2 -3670.411} C_VEL
LIN {X 0,Y 544.922,Z 287.783,A -85,B 0,C 180,E1 -3673.516,E2 -3673.516} C_VEL
LIN {X 0,Y 544.843,Z 297.29,A -85,B 0,C 180,E1 -3676.193,E2 -3676.193} C_VEL
LIN {X 0,Y 544.804,Z 299.49,A -85,B 0,C 180,E1 -3676.81,E2 -3676.81} C_VEL
LIN {X 0,Y 546.181,Z 309.407,A -85,B 0,C 180,E1 -3677.057,E2 -3677.057} C_VEL
LIN {X 0,Y 545.975,Z 322.454,A -85,B 0,C 180,E1 -3677.453,E2 -3677.453} C_VEL
LIN {X 0,Y 545.805,Z 333.473,A -85,B 0,C 180,E1 -3677.921,E2 -3677.921} C_VEL
LIN {X 0,Y 545.586,Z 345.597,A -85,B 0,C 180,E1 -3678.595,E2 -3678.595} C_VEL
LIN {X 0,Y 545.422,Z 357.082,A -85,B 0,C 180,E1 -3679.419,E2 -3679.419} C_VEL
LIN {X 0,Y 545.166,Z 367.532,A -85,B 0,C 180,E1 -3680.352,E2 -3680.352} C_VEL
LIN {X 0,Y 545.027,Z 375.986,A -85,B 0,C 180,E1 -3681.285,E2 -3681.285} C_VEL
LIN {X 0,Y 544.861,Z 384.23,A -85,B 0,C 180,E1 -3682.402,E2 -3682.402} C_VEL
LIN {X 0,Y 544.735,Z 391.616,A -85,B 0,C 180,E1 -3683.655,E2 -3683.655} C_VEL
LIN {X 0,Y 544.654,Z 396.947,A -85,B 0,C 180,E1 -3684.817,E2 -3684.817} C_VEL
LIN {X 0,Y 544.684,Z 400.892,A -85,B 0,C 180,E1 -3685.93,E2 -3685.93} C_VEL
LIN {X 0,Y 544.651,Z 403.805,A -85,B 0,C 180,E1 -3687.041,E2 -3687.041} C_VEL
LIN {X 0,Y 544.546,Z 406.182,A -85,B 0,C 180,E1 -3688.52,E2 -3688.52} C_VEL
LIN {X 0,Y 544.541,Z 407,A -85,B 0,C 180,E1 -3689.999,E2 -3689.999} C_VEL
LIN {X 0,Y 544.546,Z 406.185,A -85,B 0,C 180,E1 -3691.478,E2 -3691.478} C_VEL
LIN {X 0,Y 544.651,Z 403.812,A -85,B 0,C 180,E1 -3692.958,E2 -3692.958} C_VEL
LIN {X 0,Y 544.684,Z 400.897,A -85,B 0,C 180,E1 -3694.069,E2 -3694.069} C_VEL
LIN {X 0,Y 544.653,Z 396.951,A -85,B 0,C 180,E1 -3695.182,E2 -3695.182} C_VEL
LIN {X 0,Y 544.729,Z 391.655,A -85,B 0,C 180,E1 -3696.337,E2 -3696.337} C_VEL
LIN {X 0,Y 544.837,Z 385.472,A -85,B 0,C 180,E1 -3697.411,E2 -3697.411} C_VEL
LIN {X 0,Y 545.007,Z 377.483,A -85,B 0,C 180,E1 -3698.527,E2 -3698.527} C_VEL
LIN {X 0,Y 545.142,Z 369.34,A -85,B 0,C 180,E1 -3699.46,E2 -3699.46} C_VEL
LIN {X 0,Y 545.373,Z 359.406,A -85,B 0,C 180,E1 -3700.393,E2 -3700.393} C_VEL
LIN {X 0,Y 545.53,Z 349.603,A -85,B 0,C 180,E1 -3701.141,E2 -3701.141} C_VEL
LIN {X 0,Y 545.686,Z 338.676,A -85,B 0,C 180,E1 -3701.812,E2 -3701.812} C_VEL
LIN {X 0,Y 545.894,Z 326.12,A -85,B 0,C 180,E1 -3702.405,E2 -3702.405} C_VEL
LIN {X 0,Y 546.149,Z 313.116,A -85,B 0,C 180,E1 -3702.848,E2 -3702.848} C_VEL
LIN {X 0,Y 545.926,Z 306.399,A -85,B 0,C 180,E1 -3703.019,E2 -3703.019} C_VEL
LIN {X 0,Y 544.803,Z 299.492,A -85,B 0,C 180,E1 -3703.189,E2 -3703.189} C_VEL
LIN {X 0,Y 544.899,Z 289.088,A -85,B 0,C 180,E1 -3706.098,E2 -3706.098} C_VEL
LIN {X 0,Y 544.989,Z 279.478,A -85,B 0,C 180,E1 -3708.807,E2 -3708.807} C_VEL
LIN {X 0,Y 545.068,Z 270.037,A -85,B 0,C 180,E1 -3711.494,E2 -3711.494} C_VEL
LIN {X 0,Y 545.177,Z 260.307,A -85,B 0,C 180,E1 -3714.362,E2 -3714.362} C_VEL
LIN {X 0,Y 545.309,Z 251.179,A -85,B 0,C 180,E1 -3717.216,E2 -3717.216} C_VEL
LIN {X 0,Y 545.498,Z 241.458,A -85,B 0,C 180,E1 -3720.321,E2 -3720.321} C_VEL
LIN {X 0,Y 545.749,Z 232.988,A -85,B 0,C 180,E1 -3723.169,E2 -3723.169} C_VEL
LIN {X 0,Y 545.878,Z 225.615,A -85,B 0,C 180,E1 -3725.795,E2 -3725.795} C_VEL
LIN {X 0,Y 545.053,Z 220.594,A -85,B 0,C 180,E1 -3727.767,E2 -3727.767} C_VEL
LIN {X 0,Y 545.091,Z 220.589,A -85,B 0,C 180,E1 -3730.473,E2 -3730.473} C_VEL
LIN {X 0,Y 545.081,Z 220.591,A -85,B 0,C 180,E1 -3733.105,E2 -3733.105} C_VEL
LIN {X 0,Y 545.048,Z 220.594,A -85,B 0,C 180,E1 -3736.225,E2 -3736.225} C_VEL
LIN {X 0,Y 545.097,Z 220.589,A -85,B 0,C 180,E1 -3738.886,E2 -3738.886} C_VEL
LIN {X 0,Y 545.051,Z 220.593,A -85,B 0,C 180,E1 -3741.762,E2 -3741.762} C_VEL
LIN {X 0,Y 545.055,Z 220.595,A -85,B 0,C 180,E1 -3744.532,E2 -3744.532} C_VEL
LIN {X 0,Y 545.079,Z 220.589,A -85,B 0,C 180,E1 -3747.211,E2 -3747.211} C_VEL
LIN {X 0,Y 545.061,Z 220.592,A -85,B 0,C 180,E1 -3749.809,E2 -3749.809} C_VEL
LIN {X 0,Y 545.091,Z 220.59,A -85,B 0,C 180,E1 -3752.343,E2 -3752.343} C_VEL
LIN {X 0,Y 545.114,Z 220.586,A -85,B 0,C 180,E1 -3754.819,E2 -3754.819} C_VEL
LIN {X 0,Y 545.033,Z 220.595,A -85,B 0,C 180,E1 -3757.241,E2 -3757.241} C_VEL
LIN {X 0,Y 545.117,Z 220.587,A -85,B 0,C 180,E1 -3760.414,E2 -3760.414} C_VEL
LIN {X 0,Y 545.071,Z 220.591,A -85,B 0,C 180,E1 -3763.52,E2 -3763.52} C_VEL
LIN {X 0,Y 545.093,Z 220.589,A -85,B 0,C 180,E1 -3765.819,E2 -3765.819} C_VEL
LIN {X 0,Y 545.114,Z 220.584,A -85,B 0,C 180,E1 -3768.848,E2 -3768.848} C_VEL
LIN {X 0,Y 545.127,Z 220.585,A -85,B 0,C 180,E1 -3771.846,E2 -3771.846} C_VEL
LIN {X 0,Y 545.201,Z 220.574,A -85,B 0,C 180,E1 -3774.822,E2 -3774.822} C_VEL
LIN {X 0,Y 545.188,Z 220.576,A -85,B 0,C 180,E1 -3777.783,E2 -3777.783} C_VEL
LIN {X 0,Y 545.212,Z 220.575,A -85,B 0,C 180,E1 -3780.737,E2 -3780.737} C_VEL
LIN {X 0,Y 545.17,Z 220.58,A -85,B 0,C 180,E1 -3782.955,E2 -3782.955} C_VEL
LIN {X 0,Y 545.165,Z 220.578,A -85,B 0,C 180,E1 -3785.918,E2 -3785.918} C_VEL
LIN {X 0,Y 545.122,Z 220.585,A -85,B 0,C 180,E1 -3788.899,E2 -3788.899} C_VEL
LIN {X 0,Y 545.129,Z 220.584,A -85,B 0,C 180,E1 -3791.903,E2 -3791.903} C_VEL
LIN {X 0,Y 545.077,Z 220.59,A -85,B 0,C 180,E1 -3794.942,E2 -3794.942} C_VEL
LIN {X 0,Y 545.059,Z 220.593,A -85,B 0,C 180,E1 -3797.419,E2 -3797.419} C_VEL
LIN {X 0,Y 544.903,Z 220.614,A -85,B 0,C 180,E1 -3798.809,E2 -3798.809} C_VEL
LIN {X 0,Y 544.866,Z 221.168,A -85,B 0,C 180,E1 -3799.681,E2 -3799.681} C_VEL
LIN {X 0,Y 544.823,Z 224.66,A -85,B 0,C 180,E1 -3802.766,E2 -3802.766} C_VEL
LIN {X 0,Y 544.816,Z 227.678,A -85,B 0,C 180,E1 -3805.449,E2 -3805.449} C_VEL
LIN {X 0,Y 544.749,Z 230.176,A -85,B 0,C 180,E1 -3807.673,E2 -3807.673} C_VEL
LIN {X 0,Y 544.739,Z 233.182,A -85,B 0,C 180,E1 -3810.208,E2 -3810.208} C_VEL
LIN {X 0,Y 544.663,Z 236.207,A -85,B 0,C 180,E1 -3812.996,E2 -3812.996} C_VEL
LIN {X 0,Y 544.595,Z 239.061,A -85,B 0,C 180,E1 -3815.61,E2 -3815.61} C_VEL
LIN {X 0,Y 544.581,Z 240.443,A -85,B 0,C 180,E1 -3816.846,E2 -3816.846} C_VEL
LIN {X 0,Y 543.921,Z 240.959,A -85,B 0,C 180,E1 -3817.255,E2 -3817.255} C_VEL
LIN {X 0,Y 541.057,Z 241.91,A -85,B 0,C 180,E1 -3817.891,E2 -3817.891} C_VEL
LIN {X 0,Y 538.165,Z 242.868,A -85,B 0,C 180,E1 -3818.533,E2 -3818.533} C_VEL
LIN {X 0,Y 537.478,Z 243.398,A -85,B 0,C 180,E1 -3818.949,E2 -3818.949} C_VEL
LIN {X 0,Y 537.512,Z 244.34,A -85,B 0,C 180,E1 -3819.745,E2 -3819.745} C_VEL
LIN {X 0,Y 539.21,Z 254.596,A -85,B 0,C 180,E1 -3820.055,E2 -3820.055} C_VEL
LIN {X 0,Y 539.021,Z 267.172,A -85,B 0,C 180,E1 -3820.5,E2 -3820.5} C_VEL
LIN {X 0,Y 538.751,Z 279.029,A -85,B 0,C 180,E1 -3821.07,E2 -3821.07} C_VEL
LIN {X 0,Y 538.547,Z 289.545,A -85,B 0,C 180,E1 -3821.722,E2 -3821.722} C_VEL
LIN {X 0,Y 538.367,Z 299.977,A -85,B 0,C 180,E1 -3822.53,E2 -3822.53} C_VEL
LIN {X 0,Y 538.125,Z 310.017,A -85,B 0,C 180,E1 -3823.497,E2 -3823.497} C_VEL
LIN {X 0,Y 537.94,Z 318.542,A -85,B 0,C 180,E1 -3824.506,E2 -3824.506} C_VEL
LIN {X 0,Y 537.806,Z 325.891,A -85,B 0,C 180,E1 -3825.571,E2 -3825.571} C_VEL
LIN {X 0,Y 537.678,Z 331.852,A -85,B 0,C 180,E1 -3826.635,E2 -3826.635} C_VEL
LIN {X 0,Y 537.58,Z 336.583,A -85,B 0,C 180,E1 -3827.681,E2 -3827.681} C_VEL
LIN {X 0,Y 537.582,Z 340.187,A -85,B 0,C 180,E1 -3828.686,E2 -3828.686} C_VEL
LIN {X 0,Y 537.535,Z 342.036,A -85,B 0,C 180,E1 -3829.314,E2 -3829.314} C_VEL
LIN {X 0,Y 537.457,Z 344.666,A -85,B 0,C 180,E1 -3830.487,E2 -3830.487} C_VEL
LIN {X 0,Y 537.429,Z 346.329,A -85,B 0,C 180,E1 -3831.683,E2 -3831.683} C_VEL
LIN {X 0,Y 537.448,Z 346.999,A -85,B 0,C 180,E1 -3833.022,E2 -3833.022} C_VEL
LIN {X 0,Y 537.432,Z 346.545,A -85,B 0,C 180,E1 -3834.168,E2 -3834.168} C_VEL
LIN {X 0,Y 537.466,Z 344.928,A -85,B 0,C 180,E1 -3835.464,E2 -3835.464} C_VEL
LIN {X 0,Y 537.528,Z 341.971,A -85,B 0,C 180,E1 -3836.798,E2 -3836.798} C_VEL
LIN {X 0,Y 537.584,Z 337.455,A -85,B 0,C 180,E1 -3838.183,E2 -3838.183} C_VEL
LIN {X 0,Y 537.675,Z 332.344,A -85,B 0,C 180,E1 -3839.352,E2 -3839.352} C_VEL
LIN {X 0,Y 537.768,Z 326.365,A -85,B 0,C 180,E1 -3840.44,E2 -3840.44} C_VEL
LIN {X 0,Y 537.926,Z 319.028,A -85,B 0,C 180,E1 -3841.52,E2 -3841.52} C_VEL
LIN {X 0,Y 538.109,Z 309.618,A -85,B 0,C 180,E1 -3842.634,E2 -3842.634} C_VEL
LIN {X 0,Y 538.377,Z 300.078,A -85,B 0,C 180,E1 -3843.548,E2 -3843.548} C_VEL
LIN {X 0,Y 538.569,Z 290.396,A -85,B 0,C 180,E1 -3844.305,E2 -3844.305} C_VEL
LIN {X 0,Y 538.811,Z 278.902,A -85,B 0,C 180,E1 -3845.022,E2 -3845.022} C_VEL
LIN {X 0,Y 539.006,Z 266.361,A -85,B 0,C 180,E1 -3845.623,E2 -3845.623} C_VEL
LIN {X 0,Y 539.204,Z 253.909,A -85,B 0,C 180,E1 -3846.054,E2 -3846.054} C_VEL
LIN {X 0,Y 537.56,Z 244.284,A -85,B 0,C 180,E1 -3846.343,E2 -3846.343} C_VEL
LIN {X 0,Y 537.536,Z 240.799,A -85,B 0,C 180,E1 -3849.329,E2 -3849.329} C_VEL
LIN {X 0,Y 537.566,Z 238.099,A -85,B 0,C 180,E1 -3851.714,E2 -3851.714} C_VEL
LIN {X 0,Y 537.593,Z 235.394,A -85,B 0,C 180,E1 -3854.067,E2 -3854.067} C_VEL
LIN {X 0,Y 537.638,Z 232.726,A -85,B 0,C 180,E1 -3856.392,E2 -3856.392} C_VEL
LIN {X 0,Y 537.704,Z 229.223,A -85,B 0,C 180,E1 -3859.457,E2 -3859.457} C_VEL
LIN {X 0,Y 537.749,Z 225.807,A -85,B 0,C 180,E1 -3862.491,E2 -3862.491} C_VEL
LIN {X 0,Y 537.801,Z 222.357,A -85,B 0,C 180,E1 -3865.504,E2 -3865.504} C_VEL
LIN {X 0,Y 537.76,Z 221.525,A -85,B 0,C 180,E1 -3866.254,E2 -3866.254} C_VEL
LIN {X 0,Y 538.065,Z 221.466,A -85,B 0,C 180,E1 -3867.755,E2 -3867.755} C_VEL
LIN {X 0,Y 538.157,Z 221.451,A -85,B 0,C 180,E1 -3870.001,E2 -3870.001} C_VEL
LIN {X 0,Y 538.128,Z 221.457,A -85,B 0,C 180,E1 -3872.995,E2 -3872.995} C_VEL
LIN {X 0,Y 538.113,Z 221.457,A -85,B 0,C 180,E1 -3875.998,E2 -3875.998} C_VEL
LIN {X 0,Y 538.067,Z 221.463,A -85,B 0,C 180,E1 -3879.018,E2 -3879.018} C_VEL
LIN {X 0,Y 538.072,Z 221.463,A -85,B 0,C 180,E1 -3882.064,E2 -3882.064} C_VEL
LIN {X 0,Y 538.033,Z 221.467,A -85,B 0,C 180,E1 -3885.145,E2 -3885.145} C_VEL
LIN {X 0,Y 538.024,Z 221.467,A -85,B 0,C 180,E1 -3888.271,E2 -3888.271} C_VEL
LIN {X 0,Y 538.032,Z 221.467,A -85,B 0,C 180,E1 -3890.652,E2 -3890.652} C_VEL
LIN {X 0,Y 538.03,Z 221.466,A -85,B 0,C 180,E1 -3893.888,E2 -3893.888} C_VEL
LIN {X 0,Y 538.041,Z 221.465,A -85,B 0,C 180,E1 -3896.367,E2 -3896.367} C_VEL
LIN {X 0,Y 538.023,Z 221.469,A -85,B 0,C 180,E1 -3898.935,E2 -3898.935} C_VEL
LIN {X 0,Y 538.019,Z 221.468,A -85,B 0,C 180,E1 -3901.892,E2 -3901.892} C_VEL
LIN {X 0,Y 538.027,Z 221.468,A -85,B 0,C 180,E1 -3904.623,E2 -3904.623} C_VEL
LIN {X 0,Y 538,Z 221.473,A -85,B 0,C 180,E1 -3907.172,E2 -3907.172} C_VEL
LIN {X 0,Y 538.047,Z 221.465,A -85,B 0,C 180,E1 -3909.796,E2 -3909.796} C_VEL
LIN {X 0,Y 538.019,Z 221.47,A -85,B 0,C 180,E1 -3912.787,E2 -3912.787} C_VEL
LIN {X 0,Y 538.024,Z 221.467,A -85,B 0,C 180,E1 -3915.927,E2 -3915.927} C_VEL
LIN {X 0,Y 538.074,Z 221.461,A -85,B 0,C 180,E1 -3919.251,E2 -3919.251} C_VEL
LIN {X 0,Y 537.991,Z 221.474,A -85,B 0,C 180,E1 -3922.124,E2 -3922.124} C_VEL
LIN {X 0,Y 538.012,Z 221.469,A -85,B 0,C 180,E1 -3924.919,E2 -3924.919} C_VEL
LIN {X 0,Y 538.024,Z 221.468,A -85,B 0,C 180,E1 -3927.62,E2 -3927.62} C_VEL
LIN {X 0,Y 538.016,Z 221.471,A -85,B 0,C 180,E1 -3930.241,E2 -3930.241} C_VEL
LIN {X 0,Y 538.063,Z 221.463,A -85,B 0,C 180,E1 -3932.798,E2 -3932.798} C_VEL
LIN {X 0,Y 538.028,Z 221.466,A -85,B 0,C 180,E1 -3935.293,E2 -3935.293} C_VEL
LIN {X 0,Y 538.017,Z 221.471,A -85,B 0,C 180,E1 -3938.044,E2 -3938.044} C_VEL
LIN {X 0,Y 538.039,Z 221.465,A -85,B 0,C 180,E1 -3940.942,E2 -3940.942} C_VEL
LIN {X 0,Y 538.019,Z 221.468,A -85,B 0,C 180,E1 -3943.3,E2 -3943.3} C_VEL
LIN {X 0,Y 538.068,Z 221.462,A -85,B 0,C 180,E1 -3945.632,E2 -3945.632} C_VEL
LIN {X 0,Y 538.081,Z 221.46,A -85,B 0,C 180,E1 -3948.703,E2 -3948.703} C_VEL
LIN {X 0,Y 538.065,Z 221.464,A -85,B 0,C 180,E1 -3951.741,E2 -3951.741} C_VEL
LIN {X 0,Y 538.127,Z 221.457,A -85,B 0,C 180,E1 -3954.004,E2 -3954.004} C_VEL
LIN {X 0,Y 538.141,Z 221.452,A -85,B 0,C 180,E1 -3957.007,E2 -3957.007} C_VEL
LIN {X 0,Y 538.178,Z 221.45,A -85,B 0,C 180,E1 -3960.001,E2 -3960.001} C_VEL
LIN {X 0,Y 538.14,Z 221.453,A -85,B 0,C 180,E1 -3962.996,E2 -3962.996} C_VEL
LIN {X 0,Y 538.123,Z 221.456,A -85,B 0,C 180,E1 -3965.998,E2 -3965.998} C_VEL
LIN {X 0,Y 538.069,Z 221.462,A -85,B 0,C 180,E1 -3968.262,E2 -3968.262} C_VEL
LIN {X 0,Y 538.094,Z 221.46,A -85,B 0,C 180,E1 -3971.599,E2 -3971.599} C_VEL
LIN {X 0,Y 538.065,Z 221.465,A -85,B 0,C 180,E1 -3974.857,E2 -3974.857} C_VEL
LIN {X 0,Y 538.045,Z 221.465,A -85,B 0,C 180,E1 -3977.533,E2 -3977.533} C_VEL
LIN {X 0,Y 538.046,Z 221.467,A -85,B 0,C 180,E1 -3980.652,E2 -3980.652} C_VEL
LIN {X 0,Y 538.015,Z 221.471,A -85,B 0,C 180,E1 -3983.878,E2 -3983.878} C_VEL
LIN {X 0,Y 538.043,Z 221.467,A -85,B 0,C 180,E1 -3986.368,E2 -3986.368} C_VEL
LIN {X 0,Y 538.039,Z 221.466,A -85,B 0,C 180,E1 -3988.934,E2 -3988.934} C_VEL
LIN {X 0,Y 538.018,Z 221.47,A -85,B 0,C 180,E1 -3991.887,E2 -3991.887} C_VEL
LIN {X 0,Y 538.017,Z 221.469,A -85,B 0,C 180,E1 -3994.617,E2 -3994.617} C_VEL
LIN {X 0,Y 538.012,Z 221.47,A -85,B 0,C 180,E1 -3997.17,E2 -3997.17} C_VEL
LIN {X 0,Y 538.019,Z 221.47,A -85,B 0,C 180,E1 -3999.798,E2 -3999.798} C_VEL
LIN {X 0,Y 538.027,Z 221.467,A -85,B 0,C 180,E1 -4002.786,E2 -4002.786} C_VEL
LIN {X 0,Y 538.027,Z 221.467,A -85,B 0,C 180,E1 -4005.927,E2 -4005.927} C_VEL
LIN {X 0,Y 538.039,Z 221.466,A -85,B 0,C 180,E1 -4008.227,E2 -4008.227} C_VEL
LIN {X 0,Y 538.019,Z 221.471,A -85,B 0,C 180,E1 -4011.169,E2 -4011.169} C_VEL
LIN {X 0,Y 538.042,Z 221.643,A -85,B 0,C 180,E1 -4012.125,E2 -4012.125} C_VEL
LIN {X 0,Y 538.879,Z 226.723,A -85,B 0,C 180,E1 -4014.063,E2 -4014.063} C_VEL
LIN {X 0,Y 538.855,Z 232.957,A -85,B 0,C 180,E1 -4016.283,E2 -4016.283} C_VEL
LIN {X 0,Y 538.613,Z 240.87,A -85,B 0,C 180,E1 -4018.974,E2 -4018.974} C_VEL
LIN {X 0,Y 538.384,Z 250.02,A -85,B 0,C 180,E1 -4021.969,E2 -4021.969} C_VEL
LIN {X 0,Y 538.22,Z 259.308,A -85,B 0,C 180,E1 -4024.888,E2 -4024.888} C_VEL
LIN {X 0,Y 538.06,Z 268.552,A -85,B 0,C 180,E1 -4027.74,E2 -4027.74} C_VEL
LIN {X 0,Y 537.967,Z 277.977,A -85,B 0,C 180,E1 -4030.546,E2 -4030.546} C_VEL
LIN {X 0,Y 537.834,Z 288.875,A -85,B 0,C 180,E1 -4033.683,E2 -4033.683} C_VEL
LIN {X 0,Y 537.752,Z 298.379,A -85,B 0,C 180,E1 -4036.393,E2 -4036.393} C_VEL
LIN {X 0,Y 537.728,Z 299.225,A -85,B 0,C 180,E1 -4036.633,E2 -4036.633} C_VEL
LIN {X 0,Y 539.253,Z 309.944,A -85,B 0,C 180,E1 -4036.911,E2 -4036.911} C_VEL
LIN {X 0,Y 539.021,Z 322.114,A -85,B 0,C 180,E1 -4037.289,E2 -4037.289} C_VEL
LIN {X 0,Y 538.84,Z 333.184,A -85,B 0,C 180,E1 -4037.763,E2 -4037.763} C_VEL
LIN {X 0,Y 538.632,Z 344.199,A -85,B 0,C 180,E1 -4038.371,E2 -4038.371} C_VEL
LIN {X 0,Y 538.398,Z 355.758,A -85,B 0,C 180,E1 -4039.184,E2 -4039.184} C_VEL
LIN {X 0,Y 538.202,Z 365.514,A -85,B 0,C 180,E1 -4040.036,E2 -4040.036} C_VEL
LIN {X 0,Y 538.015,Z 374.398,A -85,B 0,C 180,E1 -4040.981,E2 -4040.981} C_VEL
LIN {X 0,Y 537.831,Z 382.999,A -85,B 0,C 180,E1 -4042.113,E2 -4042.113} C_VEL
LIN {X 0,Y 537.707,Z 389.864,A -85,B 0,C 180,E1 -4043.244,E2 -4043.244} C_VEL
LIN {X 0,Y 537.677,Z 395.363,A -85,B 0,C 180,E1 -4044.373,E2 -4044.373} C_VEL
LIN {X 0,Y 537.558,Z 399.674,A -85,B 0,C 180,E1 -4045.5,E2 -4045.5} C_VEL
LIN {X 0,Y 537.592,Z 401.956,A -85,B 0,C 180,E1 -4046.251,E2 -4046.251} C_VEL
LIN {X 0,Y 537.552,Z 403.805,A -85,B 0,C 180,E1 -4047.002,E2 -4047.002} C_VEL
LIN {X 0,Y 537.452,Z 406.181,A -85,B 0,C 180,E1 -4048.501,E2 -4048.501} C_VEL
LIN {X 0,Y 537.442,Z 407,A -85,B 0,C 180,E1 -4049.999,E2 -4049.999} C_VEL
LIN {X 0,Y 537.452,Z 406.184,A -85,B 0,C 180,E1 -4051.498,E2 -4051.498} C_VEL
LIN {X 0,Y 537.551,Z 403.812,A -85,B 0,C 180,E1 -4052.997,E2 -4052.997} C_VEL
LIN {X 0,Y 537.603,Z 400.897,A -85,B 0,C 180,E1 -4054.122,E2 -4054.122} C_VEL
LIN {X 0,Y 537.587,Z 396.951,A -85,B 0,C 180,E1 -4055.25,E2 -4055.25} C_VEL
LIN {X 0,Y 537.643,Z 392.137,A -85,B 0,C 180,E1 -4056.324,E2 -4056.324} C_VEL
LIN {X 0,Y 537.791,Z 385.471,A -85,B 0,C 180,E1 -4057.508,E2 -4057.508} C_VEL
LIN {X 0,Y 537.972,Z 377.483,A -85,B 0,C 180,E1 -4058.64,E2 -4058.64} C_VEL
LIN {X 0,Y 538.119,Z 369.295,A -85,B 0,C 180,E1 -4059.585,E2 -4059.585} C_VEL
LIN {X 0,Y 538.377,Z 359.276,A -85,B 0,C 180,E1 -4060.53,E2 -4060.53} C_VEL
LIN {X 0,Y 538.546,Z 349.393,A -85,B 0,C 180,E1 -4061.288,E2 -4061.288} C_VEL
LIN {X 0,Y 538.711,Z 338.361,A -85,B 0,C 180,E1 -4061.968,E2 -4061.968} C_VEL
LIN {X 0,Y 538.964,Z 325.758,A -85,B 0,C 180,E1 -4062.567,E2 -4062.567} C_VEL
LIN {X 0,Y 539.184,Z 312.693,A -85,B 0,C 180,E1 -4063.017,E2 -4063.017} C_VEL
LIN {X 0,Y 539.035,Z 307.354,A -85,B 0,C 180,E1 -4063.158,E2 -4063.158} C_VEL
LIN {X 0,Y 537.726,Z 299.166,A -85,B 0,C 180,E1 -4063.365,E2 -4063.365} C_VEL
LIN {X 0,Y 537.822,Z 290.127,A -85,B 0,C 180,E1 -4065.926,E2 -4065.926} C_VEL
LIN {X 0,Y 537.929,Z 279.144,A -85,B 0,C 180,E1 -4069.063,E2 -4069.063} C_VEL
LIN {X 0,Y 538.043,Z 269.096,A -85,B 0,C 180,E1 -4071.964,E2 -4071.964} C_VEL
LIN {X 0,Y 538.143,Z 260.231,A -85,B 0,C 180,E1 -4074.702,E2 -4074.702} C_VEL
LIN {X 0,Y 538.286,Z 251.608,A -85,B 0,C 180,E1 -4077.398,E2 -4077.398} C_VEL
LIN {X 0,Y 538.507,Z 243.191,A -85,B 0,C 180,E1 -4080.129,E2 -4080.129} C_VEL
LIN {X 0,Y 538.701,Z 235.399,A -85,B 0,C 180,E1 -4082.779,E2 -4082.779} C_VEL
LIN {X 0,Y 538.906,Z 227.883,A -85,B 0,C 180,E1 -4085.473,E2 -4085.473} C_VEL
LIN {X 0,Y 538.388,Z 223.374,A -85,B 0,C 180,E1 -4087.223,E2 -4087.223} C_VEL
LIN {X 0,Y 538.004,Z 221.472,A -85,B 0,C 180,E1 -4088.004,E2 -4088.004} C_VEL
LIN {X 0,Y 538.052,Z 221.466,A -85,B 0,C 180,E1 -4090.774,E2 -4090.774} C_VEL
LIN {X 0,Y 538.024,Z 221.469,A -85,B 0,C 180,E1 -4094.073,E2 -4094.073} C_VEL
LIN {X 0,Y 538.018,Z 221.469,A -85,B 0,C 180,E1 -4097.213,E2 -4097.213} C_VEL
LIN {X 0,Y 538.026,Z 221.469,A -85,B 0,C 180,E1 -4100.202,E2 -4100.202} C_VEL
LIN {X 0,Y 538.025,Z 221.469,A -85,B 0,C 180,E1 -4103.066,E2 -4103.066} C_VEL
LIN {X 0,Y 538.025,Z 221.469,A -85,B 0,C 180,E1 -4105.826,E2 -4105.826} C_VEL
LIN {X 0,Y 538.007,Z 221.47,A -85,B 0,C 180,E1 -4108.498,E2 -4108.498} C_VEL
LIN {X 0,Y 538.058,Z 221.465,A -85,B 0,C 180,E1 -4111.099,E2 -4111.099} C_VEL
LIN {X 0,Y 538.04,Z 221.468,A -85,B 0,C 180,E1 -4113.632,E2 -4113.632} C_VEL
LIN {X 0,Y 538.004,Z 221.471,A -85,B 0,C 180,E1 -4116.121,E2 -4116.121} C_VEL
LIN {X 0,Y 538.036,Z 221.468,A -85,B 0,C 180,E1 -4119.348,E2 -4119.348} C_VEL
LIN {X 0,Y 538.051,Z 221.467,A -85,B 0,C 180,E1 -4122.516,E2 -4122.516} C_VEL
LIN {X 0,Y 538.061,Z 221.463,A -85,B 0,C 180,E1 -4125.63,E2 -4125.63} C_VEL
LIN {X 0,Y 538.073,Z 221.462,A -85,B 0,C 180,E1 -4128.7,E2 -4128.7} C_VEL
LIN {X 0,Y 538.083,Z 221.463,A -85,B 0,C 180,E1 -4131.739,E2 -4131.739} C_VEL
LIN {X 0,Y 538.159,Z 221.451,A -85,B 0,C 180,E1 -4134.754,E2 -4134.754} C_VEL
LIN {X 0,Y 538.16,Z 221.451,A -85,B 0,C 180,E1 -4137.754,E2 -4137.754} C_VEL
LIN {X 0,Y 538.181,Z 221.451,A -85,B 0,C 180,E1 -4140.747,E2 -4140.747} C_VEL
LIN {X 0,Y 538.136,Z 221.457,A -85,B 0,C 180,E1 -4142.993,E2 -4142.993} C_VEL
LIN {X 0,Y 538.118,Z 221.456,A -85,B 0,C 180,E1 -4145.996,E2 -4145.996} C_VEL
LIN {X 0,Y 538.071,Z 221.462,A -85,B 0,C 180,E1 -4149.016,E2 -4149.016} C_VEL
LIN {X 0,Y 538.076,Z 221.464,A -85,B 0,C 180,E1 -4152.061,E2 -4152.061} C_VEL
LIN {X 0,Y 538.037,Z 221.468,A -85,B 0,C 180,E1 -4155.143,E2 -4155.143} C_VEL
LIN {X 0,Y 538.001,Z 221.473,A -85,B 0,C 180,E1 -4157.523,E2 -4157.523} C_VEL
LIN {X 0,Y 537.813,Z 221.497,A -85,B 0,C 180,E1 -4159.067,E2 -4159.067} C_VEL
LIN {X 0,Y 537.781,Z 223.004,A -85,B 0,C 180,E1 -4160.66,E2 -4160.66} C_VEL
LIN {X 0,Y 537.734,Z 225.705,A -85,B 0,C 180,E1 -4163.083,E2 -4163.083} C_VEL
LIN {X 0,Y 537.747,Z 228.541,A -85,B 0,C 180,E1 -4165.608,E2 -4165.608} C_VEL
LIN {X 0,Y 537.668,Z 231.261,A -85,B 0,C 180,E1 -4168.069,E2 -4168.069} C_VEL
LIN {X 0,Y 537.626,Z 234.249,A -85,B 0,C 180,E1 -4170.65,E2 -4170.65} C_VEL
LIN {X 0,Y 537.58,Z 237.17,A -85,B 0,C 180,E1 -4173.302,E2 -4173.302} C_VEL
LIN {X 0,Y 537.493,Z 240.138,A -85,B 0,C 180,E1 -4176.041,E2 -4176.041} C_VEL
LIN {X 0,Y 537.478,Z 243.398,A -85,B 0,C 180,E1 -4178.949,E2 -4178.949} C_VEL
LIN {X 0,Y 537.322,Z 244.407,A -85,B 0,C 180,E1 -4179.236,E2 -4179.236} C_VEL
LIN {X 0,Y 536.79,Z 247.047,A -85,B 0,C 180,E1 -4179.54,E2 -4179.54} C_VEL
LIN {X 0,Y 535.808,Z 251.505,A -85,B 0,C 180,E1 -4179.812,E2 -4179.812} C_VEL
LIN {X 0,Y 534.445,Z 257.464,A -85,B 0,C 180,E1 -4180.02,E2 -4180.02} C_VEL
LIN {X 0,Y 532.396,Z 267.422,A -85,B 0,C 180,E1 -4180.332,E2 -4180.332} C_VEL
LIN {X 0,Y 532.05,Z 271.071,A -85,B 0,C 180,E1 -4180.488,E2 -4180.488} C_VEL
LIN {X 0,Y 531.745,Z 282.961,A -85,B 0,C 180,E1 -4181.119,E2 -4181.119} C_VEL
LIN {X 0,Y 531.501,Z 294.278,A -85,B 0,C 180,E1 -4181.892,E2 -4181.892} C_VEL
LIN {X 0,Y 531.289,Z 304.942,A -85,B 0,C 180,E1 -4182.81,E2 -4182.81} C_VEL
LIN {X 0,Y 531.032,Z 314.55,A -85,B 0,C 180,E1 -4183.84,E2 -4183.84} C_VEL
LIN {X 0,Y 530.822,Z 323.244,A -85,B 0,C 180,E1 -4184.995,E2 -4184.995} C_VEL
LIN {X 0,Y 530.644,Z 330.776,A -85,B 0,C 180,E1 -4186.265,E2 -4186.265} C_VEL
LIN {X 0,Y 530.532,Z 336.528,A -85,B 0,C 180,E1 -4187.5,E2 -4187.5} C_VEL
LIN {X 0,Y 530.505,Z 340.24,A -85,B 0,C 180,E1 -4188.519,E2 -4188.519} C_VEL
LIN {X 0,Y 530.443,Z 343.094,A -85,B 0,C 180,E1 -4189.519,E2 -4189.519} C_VEL
LIN {X 0,Y 530.378,Z 345.163,A -85,B 0,C 180,E1 -4190.504,E2 -4190.504} C_VEL
LIN {X 0,Y 530.358,Z 346.515,A -85,B 0,C 180,E1 -4191.479,E2 -4191.479} C_VEL
LIN {X 0,Y 530.34,Z 347.298,A -85,B 0,C 180,E1 -4192.663,E2 -4192.663} C_VEL
LIN {X 0,Y 530.362,Z 347.076,A -85,B 0,C 180,E1 -4193.93,E2 -4193.93} C_VEL
LIN {X 0,Y 530.365,Z 345.665,A -85,B 0,C 180,E1 -4195.265,E2 -4195.265} C_VEL
LIN {X 0,Y 530.443,Z 343.054,A -85,B 0,C 180,E1 -4196.582,E2 -4196.582} C_VEL
LIN {X 0,Y 530.51,Z 338.762,A -85,B 0,C 180,E1 -4198.002,E2 -4198.002} C_VEL
LIN {X 0,Y 530.624,Z 332.823,A -85,B 0,C 180,E1 -4199.415,E2 -4199.415} C_VEL
LIN {X 0,Y 530.737,Z 325.973,A -85,B 0,C 180,E1 -4200.663,E2 -4200.663} C_VEL
LIN {X 0,Y 530.927,Z 318.441,A -85,B 0,C 180,E1 -4201.757,E2 -4201.757} C_VEL
LIN {X 0,Y 531.148,Z 309.251,A -85,B 0,C 180,E1 -4202.84,E2 -4202.84} C_VEL
LIN {X 0,Y 531.415,Z 300.253,A -85,B 0,C 180,E1 -4203.703,E2 -4203.703} C_VEL
LIN {X 0,Y 531.634,Z 289.273,A -85,B 0,C 180,E1 -4204.556,E2 -4204.556} C_VEL
LIN {X 0,Y 531.921,Z 277.275,A -85,B 0,C 180,E1 -4205.288,E2 -4205.288} C_VEL
LIN {X 0,Y 532.134,Z 265.667,A -85,B 0,C 180,E1 -4205.832,E2 -4205.832} C_VEL
LIN {X 0,Y 532.205,Z 253.691,A -85,B 0,C 180,E1 -4206.243,E2 -4206.243} C_VEL
LIN {X 0,Y 530.492,Z 244.666,A -85,B 0,C 180,E1 -4206.525,E2 -4206.525} C_VEL
LIN {X 0,Y 530.482,Z 241.762,A -85,B 0,C 180,E1 -4209.042,E2 -4209.042} C_VEL
LIN {X 0,Y 530.492,Z 238.962,A -85,B 0,C 180,E1 -4211.462,E2 -4211.462} C_VEL
LIN {X 0,Y 530.53,Z 236.223,A -85,B 0,C 180,E1 -4213.849,E2 -4213.849} C_VEL
LIN {X 0,Y 530.591,Z 233.536,A -85,B 0,C 180,E1 -4216.207,E2 -4216.207} C_VEL
LIN {X 0,Y 530.643,Z 230.037,A -85,B 0,C 180,E1 -4219.315,E2 -4219.315} C_VEL
LIN {X 0,Y 530.67,Z 226.525,A -85,B 0,C 180,E1 -4222.39,E2 -4222.39} C_VEL
LIN {X 0,Y 530.702,Z 223.966,A -85,B 0,C 180,E1 -4224.682,E2 -4224.682} C_VEL
LIN {X 0,Y 530.706,Z 222.384,A -85,B 0,C 180,E1 -4226.204,E2 -4226.204} C_VEL
LIN {X 0,Y 531.028,Z 222.342,A -85,B 0,C 180,E1 -4227.725,E2 -4227.725} C_VEL
LIN {X 0,Y 531.128,Z 222.326,A -85,B 0,C 180,E1 -4230.001,E2 -4230.001} C_VEL
LIN {X 0,Y 531.095,Z 222.333,A -85,B 0,C 180,E1 -4233.035,E2 -4233.035} C_VEL
LIN {X 0,Y 531.072,Z 222.335,A -85,B 0,C 180,E1 -4236.078,E2 -4236.078} C_VEL
LIN {X 0,Y 531.026,Z 222.34,A -85,B 0,C 180,E1 -4239.139,E2 -4239.139} C_VEL
LIN {X 0,Y 531.048,Z 222.337,A -85,B 0,C 180,E1 -4241.679,E2 -4241.679} C_VEL
LIN {X 0,Y 531.017,Z 222.341,A -85,B 0,C 180,E1 -4244.957,E2 -4244.957} C_VEL
LIN {X 0,Y 531.004,Z 222.344,A -85,B 0,C 180,E1 -4247.724,E2 -4247.724} C_VEL
LIN {X 0,Y 530.994,Z 222.344,A -85,B 0,C 180,E1 -4250.939,E2 -4250.939} C_VEL
LIN {X 0,Y 530.996,Z 222.342,A -85,B 0,C 180,E1 -4254.046,E2 -4254.046} C_VEL
LIN {X 0,Y 531.002,Z 222.344,A -85,B 0,C 180,E1 -4256.745,E2 -4256.745} C_VEL
LIN {X 0,Y 530.973,Z 222.347,A -85,B 0,C 180,E1 -4259.324,E2 -4259.324} C_VEL
LIN {X 0,Y 530.971,Z 222.346,A -85,B 0,C 180,E1 -4262.105,E2 -4262.105} C_VEL
LIN {X 0,Y 530.983,Z 222.347,A -85,B 0,C 180,E1 -4264.856,E2 -4264.856} C_VEL
LIN {X 0,Y 530.959,Z 222.348,A -85,B 0,C 180,E1 -4267.509,E2 -4267.509} C_VEL
LIN {X 0,Y 531.001,Z 222.343,A -85,B 0,C 180,E1 -4270.432,E2 -4270.432} C_VEL
LIN {X 0,Y 530.961,Z 222.346,A -85,B 0,C 180,E1 -4273.496,E2 -4273.496} C_VEL
LIN {X 0,Y 530.959,Z 222.35,A -85,B 0,C 180,E1 -4276.507,E2 -4276.507} C_VEL
LIN {X 0,Y 531.023,Z 222.34,A -85,B 0,C 180,E1 -4279.573,E2 -4279.573} C_VEL
LIN {X 0,Y 530.966,Z 222.347,A -85,B 0,C 180,E1 -4282.579,E2 -4282.579} C_VEL
LIN {X 0,Y 530.995,Z 222.344,A -85,B 0,C 180,E1 -4285.313,E2 -4285.313} C_VEL
LIN {X 0,Y 530.969,Z 222.348,A -85,B 0,C 180,E1 -4288.034,E2 -4288.034} C_VEL
LIN {X 0,Y 530.988,Z 222.345,A -85,B 0,C 180,E1 -4290.876,E2 -4290.876} C_VEL
LIN {X 0,Y 531.004,Z 222.342,A -85,B 0,C 180,E1 -4293.258,E2 -4293.258} C_VEL
LIN {X 0,Y 530.96,Z 222.35,A -85,B 0,C 180,E1 -4295.969,E2 -4295.969} C_VEL
LIN {X 0,Y 531.002,Z 222.344,A -85,B 0,C 180,E1 -4299.064,E2 -4299.064} C_VEL
LIN {X 0,Y 531.02,Z 222.341,A -85,B 0,C 180,E1 -4302.279,E2 -4302.279} C_VEL
LIN {X 0,Y 531.023,Z 222.34,A -85,B 0,C 180,E1 -4305.437,E2 -4305.437} C_VEL
LIN {X 0,Y 531.053,Z 222.337,A -85,B 0,C 180,E1 -4308.551,E2 -4308.551} C_VEL
LIN {X 0,Y 531.04,Z 222.338,A -85,B 0,C 180,E1 -4311.631,E2 -4311.631} C_VEL
LIN {X 0,Y 531.124,Z 222.326,A -85,B 0,C 180,E1 -4314.687,E2 -4314.687} C_VEL
LIN {X 0,Y 531.14,Z 222.327,A -85,B 0,C 180,E1 -4317.726,E2 -4317.726} C_VEL
LIN {X 0,Y 531.157,Z 222.324,A -85,B 0,C 180,E1 -4320.759,E2 -4320.759} C_VEL
LIN {X 0,Y 531.107,Z 222.329,A -85,B 0,C 180,E1 -4323.035,E2 -4323.035} C_VEL
LIN {X 0,Y 531.079,Z 222.333,A -85,B 0,C 180,E1 -4326.078,E2 -4326.078} C_VEL
LIN {X 0,Y 531.023,Z 222.342,A -85,B 0,C 180,E1 -4329.139,E2 -4329.139} C_VEL
LIN {X 0,Y 531.058,Z 222.336,A -85,B 0,C 180,E1 -4331.671,E2 -4331.671} C_VEL
LIN {X 0,Y 531.038,Z 222.34,A -85,B 0,C 180,E1 -4334.955,E2 -4334.955} C_VEL
LIN {X 0,Y 530.989,Z 222.344,A -85,B 0,C 180,E1 -4337.724,E2 -4337.724} C_VEL
LIN {X 0,Y 531.034,Z 222.339,A -85,B 0,C 180,E1 -4340.128,E2 -4340.128} C_VEL
LIN {X 0,Y 530.953,Z 222.349,A -85,B 0,C 180,E1 -4342.574,E2 -4342.574} C_VEL
LIN {X 0,Y 530.969,Z 222.349,A -85,B 0,C 180,E1 -4345.06,E2 -4345.06} C_VEL
LIN {X 0,Y 531.02,Z 222.341,A -85,B 0,C 180,E1 -4347.596,E2 -4347.596} C_VEL
LIN {X 0,Y 530.975,Z 222.346,A -85,B 0,C 180,E1 -4350.644,E2 -4350.644} C_VEL
LIN {X 0,Y 530.971,Z 222.346,A -85,B 0,C 180,E1 -4353.5,E2 -4353.5} C_VEL
LIN {X 0,Y 530.954,Z 222.348,A -85,B 0,C 180,E1 -4356.153,E2 -4356.153} C_VEL
LIN {X 0,Y 530.973,Z 222.347,A -85,B 0,C 180,E1 -4358.653,E2 -4358.653} C_VEL
LIN {X 0,Y 531.002,Z 222.342,A -85,B 0,C 180,E1 -4361.436,E2 -4361.436} C_VEL
LIN {X 0,Y 530.981,Z 222.346,A -85,B 0,C 180,E1 -4364.548,E2 -4364.548} C_VEL
LIN {X 0,Y 530.99,Z 222.344,A -85,B 0,C 180,E1 -4367.834,E2 -4367.834} C_VEL
LIN {X 0,Y 530.993,Z 222.345,A -85,B 0,C 180,E1 -4370.556,E2 -4370.556} C_VEL
LIN {X 0,Y 530.995,Z 222.527,A -85,B 0,C 180,E1 -4371.894,E2 -4371.894} C_VEL
LIN {X 0,Y 531.808,Z 227.235,A -85,B 0,C 180,E1 -4373.721,E2 -4373.721} C_VEL
LIN {X 0,Y 531.938,Z 231.743,A -85,B 0,C 180,E1 -4375.38,E2 -4375.38} C_VEL
LIN {X 0,Y 531.691,Z 240.748,A -85,B 0,C 180,E1 -4378.525,E2 -4378.525} C_VEL
LIN {X 0,Y 531.38,Z 249.879,A -85,B 0,C 180,E1 -4381.566,E2 -4381.566} C_VEL
LIN {X 0,Y 531.231,Z 259.087,A -85,B 0,C 180,E1 -4384.534,E2 -4384.534} C_VEL
LIN {X 0,Y 531.018,Z 268.335,A -85,B 0,C 180,E1 -4387.429,E2 -4387.429} C_VEL
LIN {X 0,Y 530.909,Z 277.958,A -85,B 0,C 180,E1 -4390.351,E2 -4390.351} C_VEL
LIN {X 0,Y 530.782,Z 288.607,A -85,B 0,C 180,E1 -4393.46,E2 -4393.46} C_VEL
LIN {X 0,Y 530.664,Z 298.749,A -85,B 0,C 180,E1 -4396.403,E2 -4396.403} C_VEL
LIN {X 0,Y 530.658,Z 299.133,A -85,B 0,C 180,E1 -4396.476,E2 -4396.476} C_VEL
LIN {X 0,Y 532.32,Z 310.447,A -85,B 0,C 180,E1 -4396.762,E2 -4396.762} C_VEL
LIN {X 0,Y 532.058,Z 322.998,A -85,B 0,C 180,E1 -4397.168,E2 -4397.168} C_VEL
LIN {X 0,Y 531.831,Z 334.702,A -85,B 0,C 180,E1 -4397.696,E2 -4397.696} C_VEL
LIN {X 0,Y 531.584,Z 345.664,A -85,B 0,C 180,E1 -4398.337,E2 -4398.337} C_VEL
LIN {X 0,Y 531.351,Z 356.532,A -85,B 0,C 180,E1 -4399.135,E2 -4399.135} C_VEL
LIN {X 0,Y 531.091,Z 367.066,A -85,B 0,C 180,E1 -4400.093,E2 -4400.093} C_VEL
LIN {X 0,Y 530.931,Z 375.599,A -85,B 0,C 180,E1 -4401.051,E2 -4401.051} C_VEL
LIN {X 0,Y 530.73,Z 383.922,A -85,B 0,C 180,E1 -4402.198,E2 -4402.198} C_VEL
LIN {X 0,Y 530.6,Z 391.035,A -85,B 0,C 180,E1 -4403.419,E2 -4403.419} C_VEL
LIN {X 0,Y 530.525,Z 396.78,A -85,B 0,C 180,E1 -4404.679,E2 -4404.679} C_VEL
LIN {X 0,Y 530.523,Z 400.775,A -85,B 0,C 180,E1 -4405.821,E2 -4405.821} C_VEL
LIN {X 0,Y 530.457,Z 403.722,A -85,B 0,C 180,E1 -4406.961,E2 -4406.961} C_VEL
LIN {X 0,Y 530.412,Z 405.124,A -85,B 0,C 180,E1 -4407.721,E2 -4407.721} C_VEL
LIN {X 0,Y 530.344,Z 406.735,A -85,B 0,C 180,E1 -4409.24,E2 -4409.24} C_VEL
LIN {X 0,Y 530.343,Z 406.953,A -85,B 0,C 180,E1 -4409.999,E2 -4409.999} C_VEL
LIN {X 0,Y 530.361,Z 406.127,A -85,B 0,C 180,E1 -4411.518,E2 -4411.518} C_VEL
LIN {X 0,Y 530.412,Z 405.129,A -85,B 0,C 180,E1 -4412.277,E2 -4412.277} C_VEL
LIN {X 0,Y 530.457,Z 403.727,A -85,B 0,C 180,E1 -4413.037,E2 -4413.037} C_VEL
LIN {X 0,Y 530.523,Z 400.777,A -85,B 0,C 180,E1 -4414.178,E2 -4414.178} C_VEL
LIN {X 0,Y 530.525,Z 396.778,A -85,B 0,C 180,E1 -4415.32,E2 -4415.32} C_VEL
LIN {X 0,Y 530.596,Z 391.043,A -85,B 0,C 180,E1 -4416.577,E2 -4416.577} C_VEL
LIN {X 0,Y 530.728,Z 383.915,A -85,B 0,C 180,E1 -4417.8,E2 -4417.8} C_VEL
LIN {X 0,Y 530.931,Z 375.584,A -85,B 0,C 180,E1 -4418.947,E2 -4418.947} C_VEL
LIN {X 0,Y 531.088,Z 367.044,A -85,B 0,C 180,E1 -4419.905,E2 -4419.905} C_VEL
LIN {X 0,Y 531.343,Z 356.5,A -85,B 0,C 180,E1 -4420.863,E2 -4420.863} C_VEL
LIN {X 0,Y 531.614,Z 344.8,A -85,B 0,C 180,E1 -4421.716,E2 -4421.716} C_VEL
LIN {X 0,Y 531.842,Z 332.717,A -85,B 0,C 180,E1 -4422.399,E2 -4422.399} C_VEL
LIN {X 0,Y 532.103,Z 320.33,A -85,B 0,C 180,E1 -4422.926,E2 -4422.926} C_VEL
LIN {X 0,Y 532.118,Z 308.492,A -85,B 0,C 180,E1 -4423.291,E2 -4423.291} C_VEL
LIN {X 0,Y 530.646,Z 298.761,A -85,B 0,C 180,E1 -4423.547,E2 -4423.547} C_VEL
LIN {X 0,Y 530.75,Z 289.797,A -85,B 0,C 180,E1 -4426.144,E2 -4426.144} C_VEL
LIN {X 0,Y 530.868,Z 280.187,A -85,B 0,C 180,E1 -4428.925,E2 -4428.925} C_VEL
LIN {X 0,Y 530.958,Z 270.528,A -85,B 0,C 180,E1 -4431.753,E2 -4431.753} C_VEL
LIN {X 0,Y 531.099,Z 261.269,A -85,B 0,C 180,E1 -4434.634,E2 -4434.634} C_VEL
LIN {X 0,Y 531.254,Z 252.049,A -85,B 0,C 180,E1 -4437.581,E2 -4437.581} C_VEL
LIN {X 0,Y 531.509,Z 244.231,A -85,B 0,C 180,E1 -4440.162,E2 -4440.162} C_VEL
LIN {X 0,Y 531.779,Z 235.401,A -85,B 0,C 180,E1 -4443.222,E2 -4443.222} C_VEL
LIN {X 0,Y 531.946,Z 229.086,A -85,B 0,C 180,E1 -4445.543,E2 -4445.543} C_VEL
LIN {X 0,Y 531.32,Z 224.203,A -85,B 0,C 180,E1 -4447.477,E2 -4447.477} C_VEL
LIN {X 0,Y 530.982,Z 222.348,A -85,B 0,C 180,E1 -4448.346,E2 -4448.346} C_VEL
LIN {X 0,Y 531,Z 222.343,A -85,B 0,C 180,E1 -4451.434,E2 -4451.434} C_VEL
LIN {X 0,Y 530.975,Z 222.348,A -85,B 0,C 180,E1 -4454.547,E2 -4454.547} C_VEL
LIN {X 0,Y 530.987,Z 222.347,A -85,B 0,C 180,E1 -4457.833,E2 -4457.833} C_VEL
LIN {X 0,Y 530.987,Z 222.345,A -85,B 0,C 180,E1 -4460.556,E2 -4460.556} C_VEL
LIN {X 0,Y 530.968,Z 222.347,A -85,B 0,C 180,E1 -4463.842,E2 -4463.842} C_VEL
LIN {X 0,Y 530.998,Z 222.344,A -85,B 0,C 180,E1 -4466.493,E2 -4466.493} C_VEL
LIN {X 0,Y 530.971,Z 222.347,A -85,B 0,C 180,E1 -4469.354,E2 -4469.354} C_VEL
LIN {X 0,Y 531.014,Z 222.344,A -85,B 0,C 180,E1 -4472.466,E2 -4472.466} C_VEL
LIN {X 0,Y 530.992,Z 222.345,A -85,B 0,C 180,E1 -4474.941,E2 -4474.941} C_VEL
LIN {X 0,Y 530.968,Z 222.348,A -85,B 0,C 180,E1 -4478.246,E2 -4478.246} C_VEL
LIN {X 0,Y 530.993,Z 222.344,A -85,B 0,C 180,E1 -4480.676,E2 -4480.676} C_VEL
LIN {X 0,Y 530.983,Z 222.345,A -85,B 0,C 180,E1 -4483.07,E2 -4483.07} C_VEL
LIN {X 0,Y 531.016,Z 222.34,A -85,B 0,C 180,E1 -4485.435,E2 -4485.435} C_VEL
LIN {X 0,Y 531.045,Z 222.338,A -85,B 0,C 180,E1 -4488.549,E2 -4488.549} C_VEL
LIN {X 0,Y 531.053,Z 222.339,A -85,B 0,C 180,E1 -4491.628,E2 -4491.628} C_VEL
LIN {X 0,Y 531.118,Z 222.328,A -85,B 0,C 180,E1 -4494.684,E2 -4494.684} C_VEL
LIN {X 0,Y 531.132,Z 222.327,A -85,B 0,C 180,E1 -4497.724,E2 -4497.724} C_VEL
LIN {X 0,Y 531.151,Z 222.327,A -85,B 0,C 180,E1 -4500.757,E2 -4500.757} C_VEL
LIN {X 0,Y 531.103,Z 222.332,A -85,B 0,C 180,E1 -4503.033,E2 -4503.033} C_VEL
LIN {X 0,Y 531.078,Z 222.334,A -85,B 0,C 180,E1 -4506.076,E2 -4506.076} C_VEL
LIN {X 0,Y 531.03,Z 222.339,A -85,B 0,C 180,E1 -4509.137,E2 -4509.137} C_VEL
LIN {X 0,Y 531.054,Z 222.336,A -85,B 0,C 180,E1 -4511.677,E2 -4511.677} C_VEL
LIN {X 0,Y 531.021,Z 222.342,A -85,B 0,C 180,E1 -4514.955,E2 -4514.955} C_VEL
LIN {X 0,Y 530.951,Z 222.353,A -85,B 0,C 180,E1 -4517.723,E2 -4517.723} C_VEL
LIN {X 0,Y 530.748,Z 222.378,A -85,B 0,C 180,E1 -4519.331,E2 -4519.331} C_VEL
LIN {X 0,Y 530.726,Z 225.266,A -85,B 0,C 180,E1 -4522.037,E2 -4522.037} C_VEL
LIN {X 0,Y 530.679,Z 228.644,A -85,B 0,C 180,E1 -4525.072,E2 -4525.072} C_VEL
LIN {X 0,Y 530.626,Z 231.394,A -85,B 0,C 180,E1 -4527.616,E2 -4527.616} C_VEL
LIN {X 0,Y 530.568,Z 234.714,A -85,B 0,C 180,E1 -4530.572,E2 -4530.572} C_VEL
LIN {X 0,Y 530.499,Z 237.935,A -85,B 0,C 180,E1 -4533.426,E2 -4533.426} C_VEL
LIN {X 0,Y 530.421,Z 240.772,A -85,B 0,C 180,E1 -4536.077,E2 -4536.077} C_VEL
LIN {X 0,Y 530.398,Z 244.049,A -85,B 0,C 180,E1 -4538.941,E2 -4538.941} C_VEL
LIN {X 0,Y 530.466,Z 244.79,A -85,B 0,C 180,E1 -4539.577,E2 -4539.577} C_VEL
LIN {X 0,Y 532.305,Z 255.154,A -85,B 0,C 180,E1 -4539.889,E2 -4539.889} C_VEL
LIN {X 0,Y 532.124,Z 267.347,A -85,B 0,C 180,E1 -4540.326,E2 -4540.326} C_VEL
LIN {X 0,Y 532.05,Z 271.071,A -85,B 0,C 180,E1 -4540.488,E2 -4540.488} C_VEL
LIN {X 0,Y 531.257,Z 276.504,A -85,B 0,C 180,E1 -4540.737,E2 -4540.737} C_VEL
LIN {X 0,Y 526.892,Z 288.445,A -85,B 0,C 180,E1 -4541.345,E2 -4541.345} C_VEL
LIN {X 0,Y 524.84,Z 294.967,A -85,B 0,C 180,E1 -4541.773,E2 -4541.773} C_VEL
LIN {X 0,Y 524.459,Z 298.11,A -85,B 0,C 180,E1 -4542.021,E2 -4542.021} C_VEL
LIN {X 0,Y 524.242,Z 308.214,A -85,B 0,C 180,E1 -4542.961,E2 -4542.961} C_VEL
LIN {X 0,Y 523.933,Z 317.667,A -85,B 0,C 180,E1 -4544.055,E2 -4544.055} C_VEL
LIN {X 0,Y 523.772,Z 324.595,A -85,B 0,C 180,E1 -4545.036,E2 -4545.036} C_VEL
LIN {X 0,Y 523.588,Z 330.943,A -85,B 0,C 180,E1 -4546.128,E2 -4546.128} C_VEL
LIN {X 0,Y 523.492,Z 336.105,A -85,B 0,C 180,E1 -4547.226,E2 -4547.226} C_VEL
LIN {X 0,Y 523.468,Z 340.224,A -85,B 0,C 180,E1 -4548.327,E2 -4548.327} C_VEL
LIN {X 0,Y 523.385,Z 343.247,A -85,B 0,C 180,E1 -4549.365,E2 -4549.365} C_VEL
LIN {X 0,Y 523.284,Z 346.169,A -85,B 0,C 180,E1 -4550.86,E2 -4550.86} C_VEL
LIN {X 0,Y 523.259,Z 347.637,A -85,B 0,C 180,E1 -4552.411,E2 -4552.411} C_VEL
LIN {X 0,Y 523.268,Z 347.577,A -85,B 0,C 180,E1 -4553.776,E2 -4553.776} C_VEL
LIN {X 0,Y 523.262,Z 346.469,A -85,B 0,C 180,E1 -4555.011,E2 -4555.011} C_VEL
LIN {X 0,Y 523.376,Z 344.066,A -85,B 0,C 180,E1 -4556.358,E2 -4556.358} C_VEL
LIN {X 0,Y 523.41,Z 340.183,A -85,B 0,C 180,E1 -4557.767,E2 -4557.767} C_VEL
LIN {X 0,Y 523.492,Z 336.105,A -85,B 0,C 180,E1 -4558.855,E2 -4558.855} C_VEL
LIN {X 0,Y 523.636,Z 330.667,A -85,B 0,C 180,E1 -4560.004,E2 -4560.004} C_VEL
LIN {X 0,Y 523.766,Z 324.143,A -85,B 0,C 180,E1 -4561.116,E2 -4561.116} C_VEL
LIN {X 0,Y 523.982,Z 315.678,A -85,B 0,C 180,E1 -4562.277,E2 -4562.277} C_VEL
LIN {X 0,Y 524.265,Z 306.259,A -85,B 0,C 180,E1 -4563.316,E2 -4563.316} C_VEL
LIN {X 0,Y 524.526,Z 296.554,A -85,B 0,C 180,E1 -4564.189,E2 -4564.189} C_VEL
LIN {X 0,Y 524.771,Z 286.232,A -85,B 0,C 180,E1 -4564.943,E2 -4564.943} C_VEL
LIN {X 0,Y 525.044,Z 274.108,A -85,B 0,C 180,E1 -4565.635,E2 -4565.635} C_VEL
LIN {X 0,Y 525.349,Z 261.264,A -85,B 0,C 180,E1 -4566.182,E2 -4566.182} C_VEL
LIN {X 0,Y 525.234,Z 254.361,A -85,B 0,C 180,E1 -4566.412,E2 -4566.412} C_VEL
LIN {X 0,Y 523.399,Z 245.075,A -85,B 0,C 180,E1 -4566.692,E2 -4566.692} C_VEL
LIN {X 0,Y 523.449,Z 241.203,A -85,B 0,C 180,E1 -4570.019,E2 -4570.019} C_VEL
LIN {X 0,Y 523.475,Z 238,A -85,B 0,C 180,E1 -4572.821,E2 -4572.821} C_VEL
LIN {X 0,Y 523.567,Z 235.262,A -85,B 0,C 180,E1 -4575.225,E2 -4575.225} C_VEL
LIN {X 0,Y 523.578,Z 231.611,A -85,B 0,C 180,E1 -4578.477,E2 -4578.477} C_VEL
LIN {X 0,Y 523.598,Z 228.177,A -85,B 0,C 180,E1 -4581.51,E2 -4581.51} C_VEL
LIN {X 0,Y 523.639,Z 225.568,A -85,B 0,C 180,E1 -4583.837,E2 -4583.837} C_VEL
LIN {X 0,Y 523.669,Z 223.855,A -85,B 0,C 180,E1 -4585.382,E2 -4585.382} C_VEL
LIN {X 0,Y 523.654,Z 223.262,A -85,B 0,C 180,E1 -4586.153,E2 -4586.153} C_VEL
LIN {X 0,Y 523.974,Z 223.219,A -85,B 0,C 180,E1 -4588.464,E2 -4588.464} C_VEL
LIN {X 0,Y 524.114,Z 223.202,A -85,B 0,C 180,E1 -4590.769,E2 -4590.769} C_VEL
LIN {X 0,Y 524.062,Z 223.209,A -85,B 0,C 180,E1 -4593.076,E2 -4593.076} C_VEL
LIN {X 0,Y 524.034,Z 223.212,A -85,B 0,C 180,E1 -4596.16,E2 -4596.16} C_VEL
LIN {X 0,Y 523.994,Z 223.216,A -85,B 0,C 180,E1 -4599.263,E2 -4599.263} C_VEL
LIN {X 0,Y 524.011,Z 223.214,A -85,B 0,C 180,E1 -4601.752,E2 -4601.752} C_VEL
LIN {X 0,Y 523.979,Z 223.218,A -85,B 0,C 180,E1 -4605.054,E2 -4605.054} C_VEL
LIN {X 0,Y 523.952,Z 223.221,A -85,B 0,C 180,E1 -4607.97,E2 -4607.97} C_VEL
LIN {X 0,Y 523.962,Z 223.22,A -85,B 0,C 180,E1 -4610.411,E2 -4610.411} C_VEL
LIN {X 0,Y 523.933,Z 223.223,A -85,B 0,C 180,E1 -4612.893,E2 -4612.893} C_VEL
LIN {X 0,Y 523.975,Z 223.219,A -85,B 0,C 180,E1 -4616.022,E2 -4616.022} C_VEL
LIN {X 0,Y 523.931,Z 223.224,A -85,B 0,C 180,E1 -4618.876,E2 -4618.876} C_VEL
LIN {X 0,Y 523.922,Z 223.225,A -85,B 0,C 180,E1 -4621.545,E2 -4621.545} C_VEL
LIN {X 0,Y 523.938,Z 223.222,A -85,B 0,C 180,E1 -4624.291,E2 -4624.291} C_VEL
LIN {X 0,Y 523.904,Z 223.229,A -85,B 0,C 180,E1 -4627.133,E2 -4627.133} C_VEL
LIN {X 0,Y 523.961,Z 223.219,A -85,B 0,C 180,E1 -4630.136,E2 -4630.136} C_VEL
LIN {X 0,Y 523.92,Z 223.225,A -85,B 0,C 180,E1 -4633.168,E2 -4633.168} C_VEL
LIN {X 0,Y 523.936,Z 223.222,A -85,B 0,C 180,E1 -4635.774,E2 -4635.774} C_VEL
LIN {X 0,Y 523.958,Z 223.22,A -85,B 0,C 180,E1 -4638.912,E2 -4638.912} C_VEL
LIN {X 0,Y 523.914,Z 223.225,A -85,B 0,C 180,E1 -4641.9,E2 -4641.9} C_VEL
LIN {X 0,Y 523.933,Z 223.223,A -85,B 0,C 180,E1 -4644.911,E2 -4644.911} C_VEL
LIN {X 0,Y 523.936,Z 223.223,A -85,B 0,C 180,E1 -4647.681,E2 -4647.681} C_VEL
LIN {X 0,Y 523.953,Z 223.22,A -85,B 0,C 180,E1 -4650.678,E2 -4650.678} C_VEL
LIN {X 0,Y 523.975,Z 223.22,A -85,B 0,C 180,E1 -4653.73,E2 -4653.73} C_VEL
LIN {X 0,Y 523.913,Z 223.226,A -85,B 0,C 180,E1 -4656.271,E2 -4656.271} C_VEL
LIN {X 0,Y 523.948,Z 223.221,A -85,B 0,C 180,E1 -4658.768,E2 -4658.768} C_VEL
LIN {X 0,Y 523.953,Z 223.22,A -85,B 0,C 180,E1 -4661.222,E2 -4661.222} C_VEL
LIN {X 0,Y 523.935,Z 223.223,A -85,B 0,C 180,E1 -4663.64,E2 -4663.64} C_VEL
LIN {X 0,Y 523.943,Z 223.224,A -85,B 0,C 180,E1 -4666.03,E2 -4666.03} C_VEL
LIN {X 0,Y 524.019,Z 223.214,A -85,B 0,C 180,E1 -4668.396,E2 -4668.396} C_VEL
LIN {X 0,Y 523.992,Z 223.216,A -85,B 0,C 180,E1 -4671.517,E2 -4671.517} C_VEL
LIN {X 0,Y 524.05,Z 223.209,A -85,B 0,C 180,E1 -4673.842,E2 -4673.842} C_VEL
LIN {X 0,Y 524.075,Z 223.204,A -85,B 0,C 180,E1 -4676.926,E2 -4676.926} C_VEL
LIN {X 0,Y 524.12,Z 223.201,A -85,B 0,C 180,E1 -4680.001,E2 -4680.001} C_VEL
LIN {X 0,Y 524.048,Z 223.208,A -85,B 0,C 180,E1 -4683.076,E2 -4683.076} C_VEL
LIN {X 0,Y 524.042,Z 223.209,A -85,B 0,C 180,E1 -4686.16,E2 -4686.16} C_VEL
LIN {X 0,Y 523.993,Z 223.217,A -85,B 0,C 180,E1 -4689.263,E2 -4689.263} C_VEL
LIN {X 0,Y 524.008,Z 223.214,A -85,B 0,C 180,E1 -4691.738,E2 -4691.738} C_VEL
LIN {X 0,Y 524,Z 223.216,A -85,B 0,C 180,E1 -4695.052,E2 -4695.052} C_VEL
LIN {X 0,Y 523.953,Z 223.222,A -85,B 0,C 180,E1 -4697.97,E2 -4697.97} C_VEL
LIN {X 0,Y 523.981,Z 223.218,A -85,B 0,C 180,E1 -4700.411,E2 -4700.411} C_VEL
LIN {X 0,Y 523.918,Z 223.227,A -85,B 0,C 180,E1 -4702.894,E2 -4702.894} C_VEL
LIN {X 0,Y 523.918,Z 223.225,A -85,B 0,C 180,E1 -4705.421,E2 -4705.421} C_VEL
LIN {X 0,Y 523.973,Z 223.218,A -85,B 0,C 180,E1 -4708,E2 -4708} C_VEL
LIN {X 0,Y 523.948,Z 223.224,A -85,B 0,C 180,E1 -4710.854,E2 -4710.854} C_VEL
LIN {X 0,Y 523.939,Z 223.222,A -85,B 0,C 180,E1 -4713.73,E2 -4713.73} C_VEL
LIN {X 0,Y 523.912,Z 223.226,A -85,B 0,C 180,E1 -4716.401,E2 -4716.401} C_VEL
LIN {X 0,Y 523.922,Z 223.225,A -85,B 0,C 180,E1 -4719.086,E2 -4719.086} C_VEL
LIN {X 0,Y 523.96,Z 223.221,A -85,B 0,C 180,E1 -4722.119,E2 -4722.119} C_VEL
LIN {X 0,Y 523.951,Z 223.22,A -85,B 0,C 180,E1 -4725.31,E2 -4725.31} C_VEL
LIN {X 0,Y 523.964,Z 223.219,A -85,B 0,C 180,E1 -4728.69,E2 -4728.69} C_VEL
LIN {X 0,Y 523.953,Z 223.415,A -85,B 0,C 180,E1 -4731.656,E2 -4731.656} C_VEL
LIN {X 0,Y 524.875,Z 229.113,A -85,B 0,C 180,E1 -4733.902,E2 -4733.902} C_VEL
LIN {X 0,Y 524.916,Z 235.124,A -85,B 0,C 180,E1 -4736.111,E2 -4736.111} C_VEL
LIN {X 0,Y 524.594,Z 243.437,A -85,B 0,C 180,E1 -4739.028,E2 -4739.028} C_VEL
LIN {X 0,Y 524.351,Z 252.323,A -85,B 0,C 180,E1 -4742.022,E2 -4742.022} C_VEL
LIN {X 0,Y 524.126,Z 261.512,A -85,B 0,C 180,E1 -4745.014,E2 -4745.014} C_VEL
LIN {X 0,Y 523.946,Z 270.754,A -85,B 0,C 180,E1 -4747.939,E2 -4747.939} C_VEL
LIN {X 0,Y 523.818,Z 280.148,A -85,B 0,C 180,E1 -4750.809,E2 -4750.809} C_VEL
LIN {X 0,Y 523.674,Z 291.059,A -85,B 0,C 180,E1 -4754.03,E2 -4754.03} C_VEL
LIN {X 0,Y 523.594,Z 298.709,A -85,B 0,C 180,E1 -4756.29,E2 -4756.29} C_VEL
LIN {X 0,Y 525.381,Z 310.94,A -85,B 0,C 180,E1 -4756.609,E2 -4756.609} C_VEL
LIN {X 0,Y 525.102,Z 323.808,A -85,B 0,C 180,E1 -4757.044,E2 -4757.044} C_VEL
LIN {X 0,Y 524.829,Z 336.065,A -85,B 0,C 180,E1 -4757.627,E2 -4757.627} C_VEL
LIN {X 0,Y 524.561,Z 347.165,A -85,B 0,C 180,E1 -4758.31,E2 -4758.31} C_VEL
LIN {X 0,Y 524.322,Z 358.454,A -85,B 0,C 180,E1 -4759.183,E2 -4759.183} C_VEL
LIN {X 0,Y 524.007,Z 368.471,A -85,B 0,C 180,E1 -4760.153,E2 -4760.153} C_VEL
LIN {X 0,Y 523.777,Z 378.191,A -85,B 0,C 180,E1 -4761.317,E2 -4761.317} C_VEL
LIN {X 0,Y 523.614,Z 385.935,A -85,B 0,C 180,E1 -4762.48,E2 -4762.48} C_VEL
LIN {X 0,Y 523.483,Z 393.073,A -85,B 0,C 180,E1 -4763.834,E2 -4763.834} C_VEL
LIN {X 0,Y 523.384,Z 397.821,A -85,B 0,C 180,E1 -4764.992,E2 -4764.992} C_VEL
LIN {X 0,Y 523.444,Z 401.457,A -85,B 0,C 180,E1 -4766.15,E2 -4766.15} C_VEL
LIN {X 0,Y 523.368,Z 403.326,A -85,B 0,C 180,E1 -4766.92,E2 -4766.92} C_VEL
LIN {X 0,Y 523.336,Z 404.729,A -85,B 0,C 180,E1 -4767.69,E2 -4767.69} C_VEL
LIN {X 0,Y 523.255,Z 406.339,A -85,B 0,C 180,E1 -4769.23,E2 -4769.23} C_VEL
LIN {X 0,Y 523.254,Z 406.555,A -85,B 0,C 180,E1 -4769.999,E2 -4769.999} C_VEL
LIN {X 0,Y 523.275,Z 405.727,A -85,B 0,C 180,E1 -4771.538,E2 -4771.538} C_VEL
LIN {X 0,Y 523.335,Z 404.728,A -85,B 0,C 180,E1 -4772.308,E2 -4772.308} C_VEL
LIN {X 0,Y 523.368,Z 403.322,A -85,B 0,C 180,E1 -4773.078,E2 -4773.078} C_VEL
LIN {X 0,Y 523.424,Z 400.367,A -85,B 0,C 180,E1 -4774.234,E2 -4774.234} C_VEL
LIN {X 0,Y 523.461,Z 396.365,A -85,B 0,C 180,E1 -4775.392,E2 -4775.392} C_VEL
LIN {X 0,Y 523.515,Z 391.116,A -85,B 0,C 180,E1 -4776.572,E2 -4776.572} C_VEL
LIN {X 0,Y 523.649,Z 384.734,A -85,B 0,C 180,E1 -4777.712,E2 -4777.712} C_VEL
LIN {X 0,Y 523.833,Z 376.652,A -85,B 0,C 180,E1 -4778.875,E2 -4778.875} C_VEL
LIN {X 0,Y 524.004,Z 368.418,A -85,B 0,C 180,E1 -4779.845,E2 -4779.845} C_VEL
LIN {X 0,Y 524.316,Z 358.386,A -85,B 0,C 180,E1 -4780.815,E2 -4780.815} C_VEL
LIN {X 0,Y 524.569,Z 347.477,A -85,B 0,C 180,E1 -4781.662,E2 -4781.662} C_VEL
LIN {X 0,Y 524.798,Z 335.969,A -85,B 0,C 180,E1 -4782.372,E2 -4782.372} C_VEL
LIN {X 0,Y 525.121,Z 323.703,A -85,B 0,C 180,E1 -4782.954,E2 -4782.954} C_VEL
LIN {X 0,Y 525.317,Z 310.825,A -85,B 0,C 180,E1 -4783.391,E2 -4783.391} C_VEL
LIN {X 0,Y 523.591,Z 298.325,A -85,B 0,C 180,E1 -4783.733,E2 -4783.733} C_VEL
LIN {X 0,Y 523.695,Z 288.071,A -85,B 0,C 180,E1 -4786.769,E2 -4786.769} C_VEL
LIN {X 0,Y 523.818,Z 278.474,A -85,B 0,C 180,E1 -4789.597,E2 -4789.597} C_VEL
LIN {X 0,Y 523.975,Z 268.874,A -85,B 0,C 180,E1 -4792.527,E2 -4792.527} C_VEL
LIN {X 0,Y 524.095,Z 259.713,A -85,B 0,C 180,E1 -4795.41,E2 -4795.41} C_VEL
LIN {X 0,Y 524.27,Z 250.547,A -85,B 0,C 180,E1 -4798.416,E2 -4798.416} C_VEL
LIN {X 0,Y 524.54,Z 243.071,A -85,B 0,C 180,E1 -4800.962,E2 -4800.962} C_VEL
LIN {X 0,Y 524.842,Z 234.898,A -85,B 0,C 180,E1 -4803.877,E2 -4803.877} C_VEL
LIN {X 0,Y 524.966,Z 230.252,A -85,B 0,C 180,E1 -4805.626,E2 -4805.626} C_VEL
LIN {X 0,Y 524.553,Z 226.628,A -85,B 0,C 180,E1 -4807.078,E2 -4807.078} C_VEL
LIN {X 0,Y 523.936,Z 223.225,A -85,B 0,C 180,E1 -4808.589,E2 -4808.589} C_VEL
LIN {X 0,Y 523.962,Z 223.22,A -85,B 0,C 180,E1 -4811.31,E2 -4811.31} C_VEL
LIN {X 0,Y 523.944,Z 223.223,A -85,B 0,C 180,E1 -4814.689,E2 -4814.689} C_VEL
LIN {X 0,Y 523.956,Z 223.222,A -85,B 0,C 180,E1 -4817.881,E2 -4817.881} C_VEL
LIN {X 0,Y 523.92,Z 223.226,A -85,B 0,C 180,E1 -4820.914,E2 -4820.914} C_VEL
LIN {X 0,Y 523.923,Z 223.225,A -85,B 0,C 180,E1 -4823.826,E2 -4823.826} C_VEL
LIN {X 0,Y 523.941,Z 223.224,A -85,B 0,C 180,E1 -4826.635,E2 -4826.635} C_VEL
LIN {X 0,Y 523.953,Z 223.221,A -85,B 0,C 180,E1 -4829.355,E2 -4829.355} C_VEL
LIN {X 0,Y 523.977,Z 223.219,A -85,B 0,C 180,E1 -4832.28,E2 -4832.28} C_VEL
LIN {X 0,Y 523.944,Z 223.224,A -85,B 0,C 180,E1 -4834.58,E2 -4834.58} C_VEL
LIN {X 0,Y 523.915,Z 223.225,A -85,B 0,C 180,E1 -4837.755,E2 -4837.755} C_VEL
LIN {X 0,Y 523.972,Z 223.22,A -85,B 0,C 180,E1 -4840.407,E2 -4840.407} C_VEL
LIN {X 0,Y 523.964,Z 223.22,A -85,B 0,C 180,E1 -4842.836,E2 -4842.836} C_VEL
LIN {X 0,Y 523.973,Z 223.218,A -85,B 0,C 180,E1 -4845.235,E2 -4845.235} C_VEL
LIN {X 0,Y 524.011,Z 223.215,A -85,B 0,C 180,E1 -4848.393,E2 -4848.393} C_VEL
LIN {X 0,Y 524.001,Z 223.216,A -85,B 0,C 180,E1 -4851.515,E2 -4851.515} C_VEL
LIN {X 0,Y 524.079,Z 223.205,A -85,B 0,C 180,E1 -4854.613,E2 -4854.613} C_VEL
LIN {X 0,Y 524.105,Z 223.202,A -85,B 0,C 180,E1 -4857.693,E2 -4857.693} C_VEL
LIN {X 0,Y 524.12,Z 223.202,A -85,B 0,C 180,E1 -4860.767,E2 -4860.767} C_VEL
LIN {X 0,Y 524.069,Z 223.208,A -85,B 0,C 180,E1 -4863.074,E2 -4863.074} C_VEL
LIN {X 0,Y 524.04,Z 223.211,A -85,B 0,C 180,E1 -4866.158,E2 -4866.158} C_VEL
LIN {X 0,Y 523.998,Z 223.215,A -85,B 0,C 180,E1 -4869.261,E2 -4869.261} C_VEL
LIN {X 0,Y 524.016,Z 223.213,A -85,B 0,C 180,E1 -4871.75,E2 -4871.75} C_VEL
LIN {X 0,Y 523.983,Z 223.219,A -85,B 0,C 180,E1 -4875.051,E2 -4875.051} C_VEL
LIN {X 0,Y 523.865,Z 223.235,A -85,B 0,C 180,E1 -4877.971,E2 -4877.971} C_VEL
LIN {X 0,Y 523.695,Z 223.317,A -85,B 0,C 180,E1 -4879.601,E2 -4879.601} C_VEL
LIN {X 0,Y 523.667,Z 226.15,A -85,B 0,C 180,E1 -4882.178,E2 -4882.178} C_VEL
LIN {X 0,Y 523.627,Z 228.814,A -85,B 0,C 180,E1 -4884.585,E2 -4884.585} C_VEL
LIN {X 0,Y 523.581,Z 232.166,A -85,B 0,C 180,E1 -4887.638,E2 -4887.638} C_VEL
LIN {X 0,Y 523.492,Z 235.576,A -85,B 0,C 180,E1 -4890.773,E2 -4890.773} C_VEL
LIN {X 0,Y 523.421,Z 238.813,A -85,B 0,C 180,E1 -4893.648,E2 -4893.648} C_VEL
LIN {X 0,Y 523.353,Z 241.738,A -85,B 0,C 180,E1 -4896.321,E2 -4896.321} C_VEL
LIN {X 0,Y 523.351,Z 245.218,A -85,B 0,C 180,E1 -4899.382,E2 -4899.382} C_VEL
LIN {X 0,Y 525.401,Z 255.929,A -85,B 0,C 180,E1 -4899.726,E2 -4899.726} C_VEL
LIN {X 0,Y 525.199,Z 268.895,A -85,B 0,C 180,E1 -4900.207,E2 -4900.207} C_VEL
LIN {X 0,Y 524.908,Z 280.822,A -85,B 0,C 180,E1 -4900.807,E2 -4900.807} C_VEL
LIN {X 0,Y 524.632,Z 291.559,A -85,B 0,C 180,E1 -4901.507,E2 -4901.507} C_VEL
LIN {X 0,Y 524.459,Z 298.11,A -85,B 0,C 180,E1 -4902.021,E2 -4902.021} C_VEL
LIN {X 0,Y 523.696,Z 302.773,A -85,B 0,C 180,E1 -4902.412,E2 -4902.412} C_VEL
LIN {X 0,Y 520.679,Z 310.085,A -85,B 0,C 180,E1 -4903.068,E2 -4903.068} C_VEL
LIN {X 0,Y 517.65,Z 316.878,A -85,B 0,C 180,E1 -4903.793,E2 -4903.793} C_VEL
LIN {X 0,Y 516.877,Z 320.67,A -85,B 0,C 180,E1 -4904.286,E2 -4904.286} C_VEL
LIN {X 0,Y 516.648,Z 328.655,A -85,B 0,C 180,E1 -4905.537,E2 -4905.537} C_VEL
LIN {X 0,Y 516.453,Z 335.385,A -85,B 0,C 180,E1 -4906.879,E2 -4906.879} C_VEL
LIN {X 0,Y 516.382,Z 340.349,A -85,B 0,C 180,E1 -4908.173,E2 -4908.173} C_VEL
LIN {X 0,Y 516.297,Z 344.442,A -85,B 0,C 180,E1 -4909.664,E2 -4909.664} C_VEL
LIN {X 0,Y 516.186,Z 347.102,A -85,B 0,C 180,E1 -4911.223,E2 -4911.223} C_VEL
LIN {X 0,Y 516.173,Z 347.929,A -85,B 0,C 180,E1 -4912.216,E2 -4912.216} C_VEL
LIN {X 0,Y 516.18,Z 348.09,A -85,B 0,C 180,E1 -4913.444,E2 -4913.444} C_VEL
LIN {X 0,Y 516.166,Z 347.175,A -85,B 0,C 180,E1 -4914.777,E2 -4914.777} C_VEL
LIN {X 0,Y 516.278,Z 345.05,A -85,B 0,C 180,E1 -4916.135,E2 -4916.135} C_VEL
LIN {X 0,Y 516.311,Z 341.442,A -85,B 0,C 180,E1 -4917.555,E2 -4917.555} C_VEL
LIN {X 0,Y 516.45,Z 336.163,A -85,B 0,C 180,E1 -4919.013,E2 -4919.013} C_VEL
LIN {X 0,Y 516.594,Z 330.589,A -85,B 0,C 180,E1 -4920.189,E2 -4920.189} C_VEL
LIN {X 0,Y 516.781,Z 323.678,A -85,B 0,C 180,E1 -4921.356,E2 -4921.356} C_VEL
LIN {X 0,Y 516.989,Z 315.479,A -85,B 0,C 180,E1 -4922.472,E2 -4922.472} C_VEL
LIN {X 0,Y 517.289,Z 306.507,A -85,B 0,C 180,E1 -4923.468,E2 -4923.468} C_VEL
LIN {X 0,Y 517.59,Z 296.734,A -85,B 0,C 180,E1 -4924.355,E2 -4924.355} C_VEL
LIN {X 0,Y 517.838,Z 286.34,A -85,B 0,C 180,E1 -4925.12,E2 -4925.12} C_VEL
LIN {X 0,Y 518.135,Z 274.272,A -85,B 0,C 180,E1 -4925.814,E2 -4925.814} C_VEL
LIN {X 0,Y 518.415,Z 262.63,A -85,B 0,C 180,E1 -4926.322,E2 -4926.322} C_VEL
LIN {X 0,Y 518.297,Z 255.177,A -85,B 0,C 180,E1 -4926.581,E2 -4926.581} C_VEL
LIN {X 0,Y 516.344,Z 245.413,A -85,B 0,C 180,E1 -4926.885,E2 -4926.885} C_VEL
LIN {X 0,Y 516.376,Z 241.678,A -85,B 0,C 180,E1 -4930.108,E2 -4930.108} C_VEL
LIN {X 0,Y 516.402,Z 238.867,A -85,B 0,C 180,E1 -4932.579,E2 -4932.579} C_VEL
